Omron Sysmac Studio project AGV_Mohn (Sysmac Studio 1.54.0.19, StandardProject)
(* New standard program for Dahl vehicles, equal bufferlane FB as Alpma *)

# Controller AGV_Mohn: NX1P2-9024DT1 version 1.46
Units and slaves: Node1 : NX-ECC203 (E001); Unit 2 : NX-SID800 (N3_N2); Unit 3 : NX-SID800 (N3_N3); Unit 4 : NX-SOD400 (N3_N4); Unit 5 : NX-SOD400 (N3_N5); Unit 6 : NX-SOH200 (N3_N6); Unit 7 : NX-DA3605 (N1); Unit 8 : NX-AD2203 (N3_N8); Unit 9 : NX-EC0122 (N3); Unit 1 : NX-OD3268 (N2_N1)
Task PrimaryTask (priority 4, period or condition 2000): Communication, AGV_Control, Manual_control, Navitrol, IO_List
Library MQTT 0.45_b14 0.0.45 (contents left out)
Library WewoNavitrol 1.0.2 (contents left out)

TYPE MQTTval : STRUCT
    topic : string[128];
    currentValue : STRING[512];
    sentValue : STRING[512];
END_STRUCT END_TYPE
TYPE Node_State : (STATE_Offline := 0, STATE_Online := 1, STATE_Stop := 2); END_TYPE
TYPE Navitrol_ProductionData_struct : STRUCT
    ProtocolVersion : UINT;  (* Navitrol protocol version; offset 0.0 *)
    Message_ID : UINT;  (* Message ID (3202); offset 2.0 *)
    Message_length : UDINT;  (* Message length in bytes (48 bytes); offset 4.0 *)
    OID_external : UDINT;  (* offset 8.0 *)
    OID_sent : UDINT;  (* offset 12.0 *)
    OID_active : UDINT;  (* offset 16.0 *)
    Item_type : UDINT;  (* offset 20.0 *)
    Pickup_ID : UDINT;  (* offset 24.0 *)
    Target_ID : UDINT;  (* offset 28.0 *)
    Order_status : UINT;  (* offset 32.0 *)
    In_Production : UINT;  (* offset 34.0 *)
END_STRUCT END_TYPE
TYPE Navitrol_TargetDetectionStatus_struct : STRUCT
    ProtocolVersion : UINT;  (* offset 0.0 *)
    Message_ID : UINT;  (* offset 2.0 *)
    Message_length : UDINT;  (* offset 4.0 *)
    DetectionMode : BYTE;  (* offset 8.0 *)
    TargetFount : BYTE;  (* offset 9.0 *)
    TargetReached : BYTE;  (* offset 10.0 *)
    TargetWithinSafetyDistance : BYTE;  (* offset 11.0 *)
    TargetX : REAL;  (* offset 12.0 *)
    TargetY : REAL;  (* offset 16.0 *)
    TargetAngle : REAL;  (* offset 20.0 *)
    PalletIDBeingDetected : DWORD;  (* offset 24.0 *)
    NumberOfReflectorsBeingDetected : UINT;  (* offset 28.0 *)
    FoundPallet’sID : UINT;  (* offset 30.0 *)
    ReservedField1 : UDINT;  (* offset 32.0 *)
    ReservedField2 : UDINT;  (* offset 36.0 *)
    ReservedField3 : UDINT;  (* offset 40.0 *)
    ReservedField4 : UDINT;  (* offset 44.0 *)
    ReservedField5 : UDINT;  (* offset 48.0 *)
END_STRUCT END_TYPE
TYPE Navitrol_ErrorWithLevel_Struct : STRUCT
    ProtocolVersion : UINT;  (* offset 0.0 *)
    Message_ID : UINT;  (* offset 2.0 *)
    Message_Length : UDINT;  (* offset 4.0 *)
    LevelOfHighestError : UINT;  (* offset 8.0 *)
    Reserved1 : UDINT;  (* offset 10.0 *)
    ErrorCount : UDINT;  (* offset 14.0 *)
    ErrorList : ARRAY[0..15] OF Navitrol_ErrorWithLevel_Error_Struct;  (* offset 18.0 *)
END_STRUCT END_TYPE
TYPE Navitrol_ErrorWithLevel_Error_Struct : STRUCT
    ErrorCode : UDINT;  (* offset 0.0 *)
    ErrorLevel : UDINT;  (* offset 4.0 *)
    Reserved2 : UINT;  (* offset 8.0 *)
END_STRUCT END_TYPE
TYPE Actuator_Selection : (Neither := 0, Front := 1, Rear := 2, Both := 3); END_TYPE
TYPE LED_Colour : (LED_Red := 0, LED_Orange := 1, LED_Yellow := 2, LED_Green := 3, LED_Cyan := 4, LED_Blue := 5, LED_Magenta := 6, LED_White := 7); END_TYPE
TYPE MES_Data_struct : STRUCT  (* MES data word *)
    Heartbeat_out : BOOL;  (* Feedback state of received heartbeat; offset 0.0 *)
    Idle : BOOL;  (* AGV in idle state; offset 0.1 *)
    Emergency : BOOL;  (* AGV in emergency state (stop state); offset 0.2 *)
    Obstacle : BOOL;  (* Obstacle in scanner warning; offset 0.3 *)
    Manual : BOOL;  (* AGV in manual ControlModeLift; offset 0.4 *)
    Loaded : BOOL;  (* AGV loaded or override active; offset 0.5 *)
    Actuator : BOOL;  (* Actuator active; offset 0.6 *)
    Charging : BOOL;  (* AGV being charged; offset 0.7 *)
    ObstacleStop : BOOL;  (* AGV stopped for obstacle; offset 1.0 *)
    ObstacleEstop : BOOL;  (* Object in sfety field; offset 1.1 *)
    Overhang : BOOL;  (* Overhang object sees object; offset 1.2 *)
    DoorState : BOOL;  (* Doorstatus, 1=ok; offset 1.3 *)
    ForkCollision : BOOL;  (* Fork collision status; offset 1.4 *)
    LiftWarning : BOOL;  (* Lift in warning state (unoperational); offset 1.5 *)
    LiftAuto : BOOL;  (* Lift busy with MES command; offset 1.6 *)
    DockingActive : BOOL;  (* AGV in docking state; offset 1.7 *)
END_STRUCT END_TYPE
TYPE Lift_Req_State : (Lift_Off := 0, Lift_Up := 1, Lift_Down := 2); END_TYPE
TYPE MQTT_Actuator_Request_struct : STRUCT  (* x coordinante of target *)
    Target_X : REAL;  (* y coordinante of target *)
    Target_Y : REAL;  (* Target position ID *)
    Distance : REAL;  (* Distance from target from inner and outer commands *)
    Height_Inner : INT;  (* Near target actuator height *)
    Height_Outer : INT;  (* Far from target actuator height *)
    Cargo_Required : BOOL;  (* Height_Inner needs cargo if true *)
END_STRUCT END_TYPE
TYPE Webinterface_Reply_struct : STRUCT
    State : BYTE;  (* offset 0.0 *)
    Timing : UINT;  (* offset 1.0 *)
    Version : STRING[5];  (* offset 3.0 *)
    Teaching : BYTE;  (* offset 8.0 *)
    V : REAL;  (* offset 9.0 *)
    X : REAL;  (* offset 13.0 *)
    Y : REAL;  (* offset 17.0 *)
    H : REAL;  (* offset 21.0 *)
    Level : BYTE;  (* offset 25.0 *)
    Pos_Conf : REAL;  (* offset 26.0 *)
    Error : BYTE;  (* offset 30.0 *)
    Nav_State : BYTE;  (* offset 31.0 *)
    SoC : REAL;  (* offset 32.0 *)
    Rem_Address : STRING[15];  (* offset 36.0 *)
    Mach_Type : BYTE;  (* offset 51.0 *)
    Omni_Steer : BYTE;  (* offset 52.0 *)
    Sector_Max : REAL;  (* offset 53.0 *)
    Sector_Min : REAL;  (* offset 57.0 *)
    Deadband : REAL;  (* offset 61.0 *)
    On_Route : BYTE;  (* offset 65.0 *)
    Fatal_Active : BYTE;  (* offset 66.0 *)
    Mach_ID : BYTE;  (* offset 67.0 *)
    Token : UINT;  (* offset 68.0 *)
    AgvLoaded : BYTE;  (* offset 73.0 *)
    Act_Active : BYTE;  (* offset 74.0 *)
    Act_Exist : BYTE;  (* offset 75.0 *)
END_STRUCT END_TYPE
TYPE Navitrol_SetTargetDetectionControlModeLift_struct : STRUCT
    ProtocolVersion : UINT;  (* Navitrol protocol version; offset 0.0 *)
    Message_ID : UINT;  (* Message ID (3202); offset 2.0 *)
    Message_length : UDINT;  (* Message length in bytes (48 bytes); offset 4.0 *)
    TargetDetectionControlModeLift : UINT;  (* Detection ControlModeLift, 0=off, 2=pallet detection; offset 8.0 *)
    PalletsToDetect : UDINT;  (* Bitfield (bit 0=ControlModeLiftl0, bit 1=ControlModeLiftl1, etc.); offset 10.0 *)
    NrOfReflectors : UINT;  (* Number of reflectors used in reflector docking; offset 14.0 *)
    ReflectorWidth : UINT;  (* Width of the used reflectors in mm; offset 16.0 *)
    PatternDetdist0 : UINT;  (* Distances (millimeter) between center of reflectors; offset 18.0 *)
    PatternDetdist1 : UINT;  (* Distances (millimeter) between center of reflectors; offset 20.0 *)
    PatternDetdist2 : UINT;  (* Distances (millimeter) between center of reflectors; offset 22.0 *)
    PatternDetdist3 : UINT;  (* Distances (millimeter) between center of reflectors; offset 24.0 *)
    PatternDetdist4 : UINT;  (* Distances (millimeter) between center of reflectors; offset 26.0 *)
    PatternDetdist5 : UINT;  (* Distances (millimeter) between center of reflectors; offset 28.0 *)
    PatternDetdist6 : UINT;  (* Distances (millimeter) between center of reflectors; offset 30.0 *)
    Reserved1 : UDINT;  (* Reserved bytes; offset 32.0 *)
    Reserved2 : UDINT;  (* Reserved bytes; offset 36.0 *)
    Reserved3 : UDINT;  (* Reserved bytes; offset 40.0 *)
    Reserved4 : UDINT;  (* Reserved bytes; offset 44.0 *)
END_STRUCT END_TYPE
TYPE Navitrol_SaveLogs_struct : STRUCT
    ProtocolVersion : UINT;  (* Navitrol protocol version; offset 0.0 *)
    Message_ID : UINT;  (* Message ID (1007); offset 2.0 *)
    Message_length : UDINT;  (* Message length in bytes (8 bytes); offset 4.0 *)
END_STRUCT END_TYPE
TYPE Navitrol_PauseDrive_struct : STRUCT
    ProtocolVersion : UINT;  (* Navitrol protocol version; offset 0.0 *)
    Message_ID : UINT;  (* Message ID (3006); offset 2.0 *)
    Message_length : UDINT;  (* Message length in bytes (8 bytes); offset 4.0 *)
END_STRUCT END_TYPE
TYPE Navitrol_ResumeDrive_struct : STRUCT
    ProtocolVersion : UINT;  (* Navitrol protocol version; offset 0.0 *)
    Message_ID : UINT;  (* Message ID (3007); offset 2.0 *)
    Message_length : UDINT;  (* Message length in bytes (8 bytes); offset 4.0 *)
END_STRUCT END_TYPE
TYPE Navitrol_AbortDrive_struct : STRUCT
    ProtocolVersion : UINT;  (* Navitrol protocol version; offset 0.0 *)
    Message_ID : UINT;  (* Message ID (3008); offset 2.0 *)
    Message_length : UDINT;  (* Message length in bytes (8 bytes); offset 4.0 *)
END_STRUCT END_TYPE
TYPE Navitrol_SetSpeedLimit_struct : STRUCT
    ProtocolVersion : UINT;  (* Navitrol protocol version; offset 0.0 *)
    Message_ID : UINT;  (* Message ID (3023); offset 2.0 *)
    Message_length : UDINT;  (* Message length in bytes (14 bytes); offset 4.0 *)
    SetRelease : UINT;  (* 1=set limit, 0=release limits; offset 8.0 *)
    Speed : REAL;  (* Speed in m/s; offset 10.0 *)
END_STRUCT END_TYPE
TYPE Navitrol_AbortWithData_struct : STRUCT
    ProtocolVersion : UINT;  (* Navitrol protocol version; offset 0.0 *)
    Message_ID : UINT;  (* Message ID (3033); offset 2.0 *)
    Message_length : UDINT;  (* Message length in bytes (14 bytes); offset 4.0 *)
    StatusControl : Navitrol_AbortControl_struct;  (* Bit field; offset 8.0 *)
    Reserved1 : UINT;  (* offset 10.0 *)
    Reserved2 : UINT;  (* offset 12.0 *)
END_STRUCT END_TYPE
TYPE Navitrol_AbortControl_struct : STRUCT
    EndDriveCompleted : BOOL;  (* 1=drive completed, 0=drive needs to be resend; offset 0.0 *)
    Reserved1 : BOOL;  (* offset 0.1 *)
    Reserved2 : BOOL;  (* offset 0.2 *)
    Reserved3 : BOOL;  (* offset 0.3 *)
    Reserved4 : BOOL;  (* offset 0.4 *)
    Reserved5 : BOOL;  (* offset 0.5 *)
    Reserved6 : BOOL;  (* offset 0.6 *)
    Reserved7 : BOOL;  (* offset 0.7 *)
    Reserved8 : BOOL;  (* offset 1.0 *)
    Reserved9 : BOOL;  (* offset 1.1 *)
    Reserved10 : BOOL;  (* offset 1.2 *)
    Reserved11 : BOOL;  (* offset 1.3 *)
    Reserved12 : BOOL;  (* offset 1.4 *)
    Reserved13 : BOOL;  (* offset 1.5 *)
    Reserved14 : BOOL;  (* offset 1.6 *)
    Reserved15 : BOOL;  (* offset 1.7 *)
END_STRUCT END_TYPE
TYPE Navitrol_RequestDriveCompleted_struct : STRUCT
    ProtocolVersion : UINT;  (* Navitrol protocol version; offset 0.0 *)
    Message_ID : UINT;  (* Message ID (3038); offset 2.0 *)
    Message_length : UDINT;  (* Message length in bytes (10 bytes); offset 4.0 *)
    Request : UINT;  (* 0=none, 1=docking, 2=buffer lane, 3=generic; offset 8.0 *)
END_STRUCT END_TYPE
TYPE Navitrol_SetSpeedArray_struct : STRUCT
    ProtocolVersion : UINT;  (* Navitrol protocol version; offset 0.0 *)
    Message_ID : UINT;  (* Message ID (3028); offset 2.0 *)
    Message_length : UDINT;  (* Message length in bytes (12 bytes); offset 4.0 *)
    SetRelease : UINT;  (* 1=set limit, 0=release limits; offset 8.0 *)
    Speed : UINT;  (* Array index to select; offset 10.0 *)
END_STRUCT END_TYPE
TYPE Navitrol_Errorlist_struct : STRUCT
    ProtocolVersion : UINT;  (* Navitrol protocol version; offset 0.0 *)
    Message_ID : UINT;  (* Message ID (201); offset 2.0 *)
    Message_length : UDINT;  (* Message length in bytes (variable); offset 4.0 *)
    Errcount : UDINT;  (* Amount of errors send (each is an UDINT); offset 8.0 *)
END_STRUCT END_TYPE
TYPE State_Scanner : (SCAN_Clear := 0, SCAN_Warn := 1, SCAN_Stop := 2, SCAN_eStop := 3); END_TYPE
TYPE Error_level_Enum : (Ok := 0 (* No Controller error *), Partial := 2 (* Partial fault level *), Minor := 3 (* Minor fault level *)); END_TYPE
TYPE Navitrol_RequestProductionData_struct : STRUCT
    ProtocolVersion : UINT;  (* offset 0.0 *)
    Message_ID : UINT;  (* offset 2.0 *)
    Message_length : UDINT;  (* offset 4.0 *)
    Activate_sending : UINT;  (* offset 8.0 *)
END_STRUCT END_TYPE
TYPE Pallet_Det_State : (init := 0, assent_PLC := 1, lift_Goes_To_Target := 2, counted_Pallets := 3); END_TYPE
TYPE Palletdetection_Action : (Mes_NotActive := 0, Mes_Active := 1); END_TYPE
TYPE ControlLift : (AGVusesNoLift := 0, Manual := 1, Automatic := 2 (* Controlled by MES *), SemiAutomatic := 3); END_TYPE
TYPE Lane_drop_state : (Idle_drop := 0, Active_drop := 10, Ready_to_drop := 20, Finished_drop := 30); END_TYPE
TYPE Navitrol_TargetDetectionStatusToMes_struct : STRUCT
    TargetFount : STRING[3];
    TargetReached : STRING[3];
    TargetWithinSafetyDistance : STRING[3];
    TargetX : STRING[100];
    TargetY : STRING[100];
    Angle : STRING[100];
END_STRUCT END_TYPE
TYPE MQTT_Errors_struct : STRUCT  (* x coordinante of target *)
    Error1 : STRING[256];
END_STRUCT END_TYPE
TYPE MQTT_Popup_struct : STRUCT  (* x coordinante of target *)
    ScreenLayer : INT;
    Message : STRING[256];
END_STRUCT END_TYPE
TYPE MQTT_Warnings_struct : STRUCT  (* x coordinante of target *)
    Warning1 : STRING[256];
END_STRUCT END_TYPE
TYPE stAnalogSensor : STRUCT
    RAW_VAL : INT;  (* Raw value *)
    OVR_VAL : INT;  (* Max error value *)
    UNDR_VAL : INT;  (* Min error value *)
    SP_MAX : INT;  (* Max setpoint value *)
    SP_MIN : INT;  (* Min setpoint value *)
    BWIRE_VAL : INT;  (* Broken wire value *)
    ALM_BWIRE : BOOL;  (* Broken wire detected *)
    ALM_OVR : BOOL;  (* Sensor over range *)
    ALM_OOR : BOOL;  (* Sensor out of range *)
    ALM_UNDR : BOOL;  (* Sensor under range *)
END_STRUCT END_TYPE
TYPE stBufferError : STRUCT
    CargoSensorBWIRE : BOOL;  (* Ultrasoon cargo distance sensor has broken wire *)
    BufferlaneSensorOOR : BOOL;  (* Laser distance sensor out of range *)
    LiftHeight : BOOL;  (* Lift height check when entering bufferlane *)
    StateErrorMES : BOOL;  (* Load not in range, can't be picked in lane *)
END_STRUCT END_TYPE
TYPE stBufferlane : STRUCT
    State : stBufferlaneStatus;  (* Status of bufferlane action *)
    Error : stBufferError;  (* Errors occured in bufferlane *)
END_STRUCT END_TYPE
TYPE stBufferlaneStatus : STRUCT
    ePickSTAT : Lane_pick_state;  (* Pick status *)
    eDropSTAT : Lane_drop_state;  (* Drop status *)
END_STRUCT END_TYPE
TYPE stControl : STRUCT
    NavInProduction : UINT;  (* Navitec in production *)
    NavInManual : BOOL;  (* Navitec in manual state *)
    NavTargetReached : UINT;  (* Navitrol reached target status *)
    NavCust1 : REAL;  (* Special route property in Navithor Tools *)
    NavCust2 : REAL;  (* Special route property in Navithor Tools *)
    NavCust3 : REAL;  (* Special route property in Navithor Tools *)
    NavCust4 : REAL;  (* Special route property in Navithor Tools *)
    NavCust5 : REAL;  (* Special route property in Navithor Tools *)
    BufferAction : INT;  (* Pick or drop action determined by MES *)
    BufferReleaseHold : BOOL;  (* Release AGV determined by MES *)
    AGVloaded : BOOL;  (* AGV is loaded *)
    AGVdir : BOOL;  (* 0 = fwdDirection of AGV *)
    AGVstandstill : BOOL;  (* AGV standstill *)
    CargoRequired : BOOL;  (* Cargo required *)
    ClientConnected : BOOL;  (* MQTT client connected *)
    ResetButton : BOOL;  (* Reset errors by operator *)
END_STRUCT END_TYPE
TYPE Lane_pick_state : (Idle_pick := 0, Active_pick := 10, Ready_to_lower_lift_pick := 20, Ready_to_pick := 30, Finished_pick := 40); END_TYPE
TYPE Lane_state_MES : (Idle := 0, Picking_Active := 10, Picking_Drive_In := 20, Picking := 30, Picking_Finished := 40, Dropping_Active := 50, Dropping := 60, Dropping_Finished := 70); END_TYPE
TYPE stClampError : STRUCT  (* Error handling for customer Alpma *)
    ClampSensorBWIRE : BOOL;  (* One of clamp sensor broken wire *)
END_STRUCT END_TYPE
TYPE stOverhang : STRUCT
    UsesPF : BOOL;  (* Pepperl and Fuchs sensor *)
    UsesSICK : BOOL;  (* SICK sensor *)
    DetectedPF : BOOL;  (* PFuchs sensor detect signal *)
    DetectedSICK : BOOL;  (* SICK sensor detect signal *)
END_STRUCT END_TYPE
TYPE stClamp : STRUCT
    IO : stClampIO;
    CargoClamped : BOOL;  (* Cargo is clamped *)
END_STRUCT END_TYPE
TYPE stClampIO : STRUCT
    Load1 : BOOL;  (* Switch NC sensor 1 in clamp *)
    Load2 : BOOL;  (* Switch NC sensor 2 in clamp *)
    Attached : BOOL;  (* Feedback clamp is attached *)
END_STRUCT END_TYPE

VAR_GLOBAL
    ClientConnected : BOOL;  (* MQTT client connected *)
    Mqtt_values : ARRAY[0..32] OF MQTTval;  (* Address:; [0] will; [1] liftHeight; [2] load; [3] safety; [4] eStopButton; [5] scanner1; [6] scanner2; [7] scanner3; [8] docking; [9] manualDrive; [10] manualLift; [11] brakeRelease; [12] charging; [13] cancelRequest; [14] cancelConfirm; [15] forkCollision *)
    Stations_State : Node_State;
    MES_State : Node_State;
    MES_Target : MQTT_Actuator_Request_struct;  (* MES actuator request by MQTT *)
    MES_PalletDetection : Palletdetection_Action;
    AGVusesRS232 : BOOL;
    AGV_Init : UINT := 0;  (* A runonce function to load values into registers *)
    Dir_Encoder1 : BOOL;  (* 0=Forward *)
    Brake_Override_Switch : BOOL;  (* Manual override switch *)
    Manual_ControlModeLift : BOOL;
    AGV_Docking : BOOL;  (* Safety reports AGV in docking ControlModeLift; at ECAT://node#[1,1]/Docking_Active *)
    Reset_Flag : BOOL;  (* Reset function called *)
    Navitrol_Tag : Navitrol_Status_TagV4_sec_struct;  (* Navitrol tag status message *)
    ToChargerTag : UDINT;  (* Virtual tag id *)
    ChargerTag : UDINT;  (* Tag ID for chargers *)
    Standstill : BOOL;  (* DoubleCheck for 0 speed *)
    Charge_Relay : BOOL;  (* Enable contact power *)
END_VAR
VAR_GLOBAL CONSTANT
    RS232_BoardID : _sOPTBOARD_ID := (SlotNo := 1, IPAdr := [5(16#0)]);  (* Board ID *)
END_VAR
VAR_GLOBAL
    ENC1_Dir_Raw : BOOL;  (* Value from enocder slice; at ECAT://node#[1,9]/Ch1 Encoder Counter Status/Ch1 Count Direction Flag *)
    ENC1_Dir : BOOL;
    Scanner_Stop : BOOL;  (* object in safety field *)
    Pump_Ok : BOOL;  (* Pump system ok *)
    Estop_Out : BOOL;  (* E-Stop has been pressed and not yet reset; at ECAT://node#[1,1]/Estop_Out *)
    Motor_Ok : BOOL;  (* Motor power active *)
    PLC_status : PLC_Status_Struct;  (* PLC status message *)
    Motor_Power_1 : BOOL;  (* Power relay 1 coil; at ECAT://node#[1,6]/Standard Input 1st Byte/So00 Monitor Value *)
    Motor_Power_2 : BOOL;  (* Power relay 2 coil; at ECAT://node#[1,6]/Standard Input 1st Byte/So01 Monitor Value *)
    Pump_Power_1 : BOOL;
    Pump_Power_2 : BOOL;
    Warning_ActuatorTime : BOOL;  (* Lift action took too long *)
    Brake_release : BOOL;  (* Brakes manual release *)
    ENC1_Speed : REAL;  (* Encoder speed in m/s *)
    Navitrol_status : Navitrol_Status_Struct;  (* Navitrol status message *)
    RotPerMin : REAL;  (* Encoder rotation per minute *)
    ENC1_Rate : UDINT;  (* Measured speed in pulses; at ECAT://node#[1,9]/Ch1 Pulse Rate *)
    AGVusesActuator : BOOL;  (* True makes sure status message is updated in the actuator section *)
    AGVusesSteering : BOOL;  (* AGV uses a steering wheel to manouver, set to 0 for differential drive *)
    AGVhasHandheld : BOOL;  (* AGV can be controlled using remote control *)
    AnalogLoad : BOOL;  (* AGV uses an analog sensor for load detection *)
    AGV_MaxSpeed : REAL;  (* Max speed in m/s *)
    NavitrolArrayLimit : BOOL;  (* Use navitrol speed array *)
    NavitrolSpeedLimit : BOOL;  (* use navitrol speed limit *)
END_VAR
VAR_GLOBAL RETAIN
    MachineID : INT;  (* Machine ID from navithor & MES *)
END_VAR
VAR_GLOBAL
    Navitrol_IP : STRING[256] := '';  (* Navigation controller *)
    Navitrol_TX_Port : UINT := 0;  (* TCP server port *)
    Navitrol_RX_Port : UINT := 0;  (* TCP listen port *)
    Navitrol_ManualSection_Enabled : BOOL;  (* Send manual section to Navitrol *)
    Navitrol_ErrorSection_Enabled : BOOL;  (* Send error messages to Navitrol *)
    Navitrol_InputSection_Enabled : BOOL;  (* Send input section to Navitrol *)
    Navitrol_LaserSection_Enabled : BOOL;  (* Send laser scanner section to Navitrol *)
    RequestGeneralSection : BOOL;  (* Ask for the general section (ID=1) from navitrol status *)
    RequestHoldSection : BOOL;  (* Ask for the hold section (ID=2) from navitrol status *)
    RequestVirtualTagSection : BOOL;  (* Ask for the virtual tag section (ID=3) from navitrol status *)
    RequestComingGoingSection : BOOL;  (* Ask for the 'Coming from, going to' section (ID=4) from navitrol status *)
    RequestCustomAtributeSection : BOOL;  (* Ask for the custom atribute section (ID=6) from navitrol status *)
    RequestWarningSection : BOOL;  (* Ask for the warning zone section (ID=7) from navitrol status *)
    RequestOutputsSection : BOOL;  (* Ask for the output section (ID=8) from navitrol status *)
    RequestBatterySection : BOOL;
    RequestDriveInfoSection : BOOL;
    RequestDistanceInfoSection : BOOL;
    NrOfSections : UINT := 0;  (* Amount of requested sections *)
    Sections : ARRAY[1..10] OF UINT;  (* Array for requested sections *)
    Navitrol_ActSection_Enabled : BOOL;  (* Send actuator section to Navitrol *)
    PLC_act : PLC_Act_Sec_Struct;
    Lift_Bot_Pos : BOOL;
    Lift_Top_Pos : BOOL;
    MessageLength : UDINT;  (* Tx message length in bytes *)
    RequestSteeringAngleSection : BOOL;  (* Ask for the steering angle section (ID=9) from navitrol status, sets with AGVusesSteering *)
    ActuatorAction : BOOL;  (* Remove power from drive motor *)
    Reset_Button : BOOL;  (* Reset input button *)
    HMI_Input0 AT %0.00 : BOOL;  (* RESET; published *)
    Safe_Reset_button : BOOL;  (* Reset button status for safety; at ECAT://node#[1,1]/Reset_Button *)
    Rel_Spd_Nav1 : INT;  (* Navitrol relative vehicle speed; at ECAT://node#[1,1]/Speed_Nav *)
    Abs_Spd_Enc1 : INT;  (* Encoder 1 absolute wheel speed *)
    Steering_Cos_Rad : REAL;  (* Cosine from target angle in Rad *)
    Navitrol_Steer : Navitrol_Status_Steering_Sec_Struct;
    Rel_Spd_Enc1 : INT;  (* Encoder relative vehicle speed; at ECAT://node#[1,1]/Speed_Enc_Rel *)
    Comp_Rel_Spd_Enc1 : INT;  (* Compensated relative enocder speed; at ECAT://node#[1,1]/Speed_Enc *)
    Dir_Navitrol1 : BOOL;  (* 0=Forward *)
    OptionalFieldReq : INT;  (* Special field selection; at ECAT://node#[1,1]/OptionalFieldReq *)
    Navitrol_SpeedUpdate : BOOL;  (* Navitrol should use a different speed setting *)
    SetNavitrolSpeedLimit : BOOL;  (* Send true to use speed limiter *)
    SpeedArray : UINT;  (* Array selection (0..4) *)
    SpeedLimit : REAL;  (* Max speed in m/s for limiter message *)
    Board_Detected : BOOL;  (* Sensor detects fork board *)
    Scanner_Slowdown : BOOL;  (* object in slowdown field *)
    Safe_Scanner_Slowdown : BOOL;  (* Slowdown to 0 field status to safety; at ECAT://node#[1,1]/Scanner_slowdown *)
    Error_Fork_Object : BOOL;  (* Fork object detection triggered *)
    Estop_requested : BOOL;  (* Request uncontrolled stop from safety; at ECAT://node#[1,1]/Estop_Request *)
    Scan1_Warn : BOOL;  (* Front right warning field *)
    Scanner_Warning : BOOL;  (* object in outer field *)
    Warning_SlowedByObstacle : BOOL;  (* Object detected in outer field while moving *)
    Scan1_Slow : BOOL;  (* Front right stop field *)
    Warning_StoppedByObstacle : BOOL;  (* Object detected in slowdown field *)
    Warning_Active : BOOL;  (* A warning is active *)
    Error_Active : BOOL;  (* A error is active *)
    HMI_Input7 AT %0.07 : BOOL;  (* Buzzer button *)
    Buzzer : BOOL;  (* Audio output *)
    PLC_Navitrol_laserscanners : PLC_Navitrol_Status_laserscanner_struct;  (* PLC to Navitrol laserscanner section *)
    Warning_StopNavitrol : BOOL;  (* AGV keeps navitrol stopped *)
    Right_door_closed : BOOL;  (* Cover is closed *)
    Left_door_closed : BOOL;  (* Cover is closed *)
    Front_door_closed : BOOL;  (* Cover is closed *)
    Warning_Cover_Open : BOOL;  (* One or more covers are not closed *)
    Lift_pump : BOOL;  (* Enables hydraulic pump *)
    StopRequest : BOOL;  (* Request controlled stop from safety PLC; at ECAT://node#[1,1]/StopRequest *)
    Update_Navitrol : BOOL;  (* Update navitrol asap *)
    LED_Reset : BOOL;  (* Indicator light *)
    LED_Left : BOOL;  (* Disable left LED bar *)
    LED_Mid1 : BOOL;  (* Disable middle-left LED bar *)
    LED_Right : BOOL;  (* Disable right LED bar *)
    LED_Mid2 : BOOL;  (* Disable middle-right LED bar *)
    Navitrol_DriveInfo : Navitrol_Status_DriveorderInfo_sec_struct;  (* Driveinfo section *)
    Blue_spot1 : BOOL;  (* Front facing Bluespot *)
    Blue_spot2 : BOOL;  (* Rear facing Bluespot *)
    Manual_Navitrol : BOOL;  (* Navitrol in manual state *)
    LED_R : INT;
    LED_G : INT;
    LED_B : INT;
    Navitrol_Battery : Navitrol_Status_Battery_struct;  (* Battery status from navitrol *)
    MES_Out_Ack AT %20.0 : BOOL;  (* Heartbeat that should change every second *)
    MES_Battery AT %20.8 : SINT;
    MES_InProd AT %20.1 : BOOL;  (* AGV in production in Navithor *)
    MES_AGVstatus AT %253 : MES_Data_struct;  (* Word for AGV status *)
    Manual_mode_switch : BOOL;  (* Manual ControlModeLift hardware switch *)
    Warning_NoPallet : BOOL;
    Warning_Lift_NOK : BOOL;  (* Lift sensor not in valid range *)
    MES_Height_Act AT %254 : UINT;  (* Actual height feedback for MES *)
    MES_MID0 AT %20.2 : BOOL;
    MES_MID1 AT %20.3 : BOOL;
    HMI_Input4 AT %0.04 : BOOL;  (* Force docking Mode; published *)
    HMI_Output0 AT %2.00 : BOOL;  (* Show RESET; published *)
    HMI_Output7 AT %2.07 : BOOL;  (* Lid; published *)
    HMI_Input3 AT %0.03 : BOOL;  (* Brake release; published *)
    HMI_Input6 AT %0.06 : BOOL;  (* Silent Mode; published *)
    HMI_Output6 AT %2.06 : BOOL;  (* Silent state; published *)
    HMI_Output9 AT %2.09 : BOOL;  (* Docking state; published *)
    HMI_Output5 AT %2.05 : BOOL;  (* HMI red fork sensors *)
    HMI_Output4 AT %2.04 : BOOL;  (* HMI all clear *)
    HMI_Int2 AT %12 : INT;  (* Front scanner; published *)
    HMI_Int3 AT %13 : INT;  (* Rear Scanner; published *)
    HMI_Int4 AT %14 : INT;  (* Estop state; published *)
    HMI_LED AT %3 : INT;  (* LED colour; published *)
    HMI_Int0 AT %10 : INT;  (* Battery level %; published *)
    HMI_Int1 AT %11 : INT;  (* Position confidence %; published *)
    Scan1_Stop : BOOL;  (* Front right safety scanner status; at ECAT://node#[1,2]/Standard Input 1st Word/Si02 Logical Value *)
    Estop_Channel1 : BOOL;  (* Emergency stop status; at ECAT://node#[1,2]/Standard Input 1st Word/Si00 Logical Value *)
    RM_Estop : BOOL;  (* Remote E-stop  state *)
    HMI_Int5 AT %15 : INT;  (* Machine ID; published *)
    HMI_Int6 AT %16 : INT;  (* HMI height feedback; published *)
    HMI_Int9 AT %19 : INT;  (* Lift max value; published *)
    Error_MotorPower : BOOL;  (* Error in motor feedback; at ECAT://node#[1,1]/Error_MotorEDM *)
    Error_PumpPower : BOOL;  (* Error in pump feedback *)
    Error_Navitrol : BOOL;  (* Navitrol reports an error *)
    Fork_bump_det_1 : BOOL;  (* Fork tip sensor *)
    Fork_bump_det_2 : BOOL;  (* fork tip sensor *)
    WarningCount : USINT := 0;  (* Amount of active warnings counter *)
    PLC_Warn_Array : array[0..4] of PLC_Warn_struct;  (* PLC warning list to send to Navitrol *)
    Warning_TableLift_Without_load : BOOL;  (* Table has been ordered to rise without load present *)
    Warning_TableDrop_Without_Load : BOOL;  (* Table has been ordered to lower without load *)
    Warning_TableLoad_Lost : BOOL;  (* Lost tabel load while lift was high *)
    HMI_Warning1 AT %135 : UINT;  (* Error code for 1st warning; published *)
    HMI_WarningText1 AT %140 : INT;
    HMI_Warning2 AT %136 : UINT;  (* Error code for 2nd warning; published *)
    HMI_WarningText2 AT %144 : INT;
    HMI_Warning3 AT %137 : UINT;  (* Error code for 3rd warning; published *)
    HMI_WarningText3 AT %148 : INT;
    HMI_Warning4 AT %138 : UINT;  (* Error code for 4th warning; published *)
    HMI_WarningText4 AT %152 : INT;
    HMI_Warning5 AT %139 : UINT;  (* Error code for 5th warning; published *)
    HMI_WarningText5 AT %156 : INT;
    ErrorCount : USINT := 0;  (* Amount of active errors counter *)
    Docking_error : BOOL;
    PLC_Error_Array : array[0..4] of PLC_Error_struct;  (* PLC error list to send to Navitrol *)
    SpeedError : BOOL;  (* Error in safety speedcheck; at ECAT://node#[1,1]/SpeedErrorStandard *)
    ErrorIndex : USINT;
    HMI_Error1 AT %50 : UINT;  (* Error code for 1st error; published *)
    HMI_ErrorText1 AT %60 : INT;
    HMI_Error2 AT %51 : UINT;  (* Error code for 2nd error; published *)
    HMI_ErrorText2 AT %64 : INT;
    HMI_Error3 AT %52 : UINT;  (* Error code for 3rd error; published *)
    HMI_ErrorText3 AT %68 : INT;
    HMI_Error4 AT %53 : UINT;  (* Error code for 4th error; published *)
    HMI_ErrorText4 AT %72 : INT;
    HMI_Error5 AT %54 : UINT;  (* Error code for 5th error; published *)
    HMI_ErrorText5 AT %76 : INT;
    Lift_valve : BOOL;  (* Opens hydraulic lift valve *)
    Lift_Prop_Speed : INT;  (* Proportional speed to lift controller *)
    HMI_Input5 AT %0.05 : BOOL;  (* Lift override; published *)
    HMI_Input1 AT %0.01 : BOOL;  (* UP; published *)
    HMI_Input2 AT %0.02 : BOOL;  (* DOWN; published *)
    HMI_Int7 AT %17 : INT;  (* Manual set height; published *)
    Rm_ManDown : BOOL;
    Rm_ManUp : BOOL;
    InProd : BOOL;  (* AGV in production *)
    Navitrol_act : Navitrol_Status_Act_Sec_Struct;
    PumpPower : BOOL;  (* Pump has power; at ECAT://node#[1,1]/PumpPower *)
    Load1 : BOOL;  (* Load sensor 1 *)
    Load2 : BOOL;  (* Load sensor 2 *)
    HMI_Int8 AT %18 : INT;  (* Lift min value; published *)
    N3_N3_Si02 : BOOL;  (* End stop switch for lift; at ECAT://node#[1,3]/Standard Input 1st Word/Si02 Logical Value *)
    Warning_Cargo_NOK : BOOL;  (* Lift action with invalid cargo *)
    TCPReady : BOOL;  (* TCP communication available *)
    RequestDriveReady : BOOL;  (* Target reached *)
    DriveType : UINT;  (* Request ready tpe *)
    Lift_Height_Raw : INT;  (* Encoder value; at ECAT://node#[1,8]/Ch1 Analog Input Value *)
    Navitrol_DistanceInfo : Navitrol_Status_DistanceToTarget_sec_struct;  (* Driveorder information *)
    MES_Height_Req AT %21 : UINT;  (* Desired height from MES *)
    Navitrol_FromTo : Navitrol_Status_FromTo_Sec_struct;
    RM_FR1 : INT;  (* Remote Forward/Reverse channel 1 *)
    RM_Center : INT;  (* Remote center tap *)
    RM_LR1 : INT;  (* Remote Left/Right channel 1 *)
    IPC_Driving_active AT %252 : BOOL;  (* Activate HTTP requests; published *)
    IPC_Driving_x AT %250 : INT;  (* x value to IPC; published *)
    IPC_Driving_y AT %251 : INT;  (* y value to IPC; published *)
    RM_Switch : INT;  (* Remote joystick switch (digital) *)
    RemoteButtonPressed : BOOL;  (* Joystick button is pressed *)
    RM_Dwn : INT;  (* Remote lift down button *)
    RM_Up : INT;  (* Remote lift up button *)
    Remote_Present : BOOL;
    HMI_Input10 AT %0.10 : BOOL;  (* Activate Remote control; published *)
    Error_Remote : BOOL := False;  (* Center tap voltage too low, no remote connected *)
    Navitrol_gen : Navitrol_Status_General_Sec_Struct;  (* Navitrol general message *)
    PLC_Navitrol_input : Navitrol_Status_inputs_struct;  (* PLC to navitrol input values *)
    NumBytes : UINT := 0;  (* Number of bytes in virtual IO (max32) *)
    NumInts : UINT := 0;  (* Number of integers in virtual IO (max32) *)
    NumFloats : UINT := 0;  (* Number of floats in virtual IO (max32) *)
    Navitrol_RemoteControlSection_Enabled : BOOL;
    Navitrol_Drivecontrol_Enabled : BOOL;
    Navitrol_PLC_Battery_Enabled : BOOL;
    NavitrolPause : BOOL;  (* Request navitrol to pause drive *)
    NavitrolResume : BOOL;  (* Request navitrol to resume drive order *)
    SendTargetDetectionSettings : BOOL;  (* send message 3202 to navitrol *)
    NavitrolAbort : BOOL;  (* Request navitrol to abort drive *)
    SafetyFieldNumber : INT;  (* Active field ID; at ECAT://node#[1,1]/ActiveFieldID *)
    Scan2_Stop : BOOL;  (* Front left safety scanner status; at ECAT://node#[1,2]/Standard Input 1st Word/Si04 Logical Value *)
    Motor_EDM_1 : BOOL;  (* Power relay 1 feedback; at ECAT://node#[1,3]/Standard Input 2nd Byte/Si00 Status *)
    Motor_EDM_2 : BOOL;  (* Power relay 2 feedback; at ECAT://node#[1,3]/Standard Input 2nd Byte/Si01 Status *)
    Scan3_Stop : BOOL;  (* Fork safety scanner status; at ECAT://node#[1,2]/Standard Input 1st Word/Si06 Logical Value *)
    Zone1 : BOOL;  (* Scanner zone select 1; at ECAT://node#[1,4]/Standard Input 1st Byte/So00 Monitor Value *)
    zone2 : BOOL;  (* Scanner zone select 2; at ECAT://node#[1,4]/Standard Input 1st Byte/So01 Monitor Value *)
    Zone3 : BOOL;  (* Scanner zone select 3; at ECAT://node#[1,4]/Standard Input 1st Byte/So02 Monitor Value *)
    Zone4 : BOOL;  (* Scanner zone select 4; at ECAT://node#[1,4]/Standard Input 1st Byte/So03 Monitor Value *)
    Zone5 : BOOL;  (* Scanner zone select 5; at ECAT://node#[1,5]/Standard Input 1st Byte/So00 Monitor Value *)
    STO_out : BOOL;  (* Safety torque off signal; at ECAT://node#[1,5]/Standard Input 1st Byte/So02 Monitor Value *)
    BufferLaneSensorDistance : INT;
    Load_Distance : INT;  (* Distance to load; at ECAT://node#[1,8]/Ch2 Analog Input Value *)
    Scan3_Warn : BOOL;  (* Fork warning field *)
    Scan3_slow : BOOL;  (* Fork stop field *)
    Lift_Control_Dir : BOOL;  (* Direction input for lift controller *)
    Indicator_Left : BOOL;  (* Route takes a left turn *)
    Indicator_Right : BOOL;  (* Route takes a right turn *)
    K11 : BOOL;  (* Pump flow direction *)
    K12 : BOOL;  (* Pump flow direction *)
    HMI_Manual AT %2.10 : BOOL;  (* Provide HMI if AGV is in manual state *)
    HMI_Int10 AT %24 : INT;  (* Battery state (enum); published *)
    HMI_MessageCount AT %26 : INT;  (* Total number of warning and error messages; published *)
    SafetyStopped : BOOL;  (* Safety is cutting power; at ECAT://node#[1,1]/SafetyStop *)
    AgvLoaded : BOOL;  (* Object loaded *)
    Scanner1_State : State_Scanner;
    Scanner2_State : State_Scanner;
    Scanner3_State : State_Scanner;
    I00 : BOOL;  (* NX1 input 0; at BuiltInIO://cpu/#0/Input_Bit_00 *)
    I01 : BOOL;  (* NX1 input 1; at BuiltInIO://cpu/#0/Input_Bit_01 *)
    I02 : BOOL;  (* NX1 input 2; at BuiltInIO://cpu/#0/Input_Bit_02 *)
    I03 : BOOL;  (* NX1 input 3; at BuiltInIO://cpu/#0/Input_Bit_03 *)
    I04 : BOOL;  (* NX1 input 4; at BuiltInIO://cpu/#0/Input_Bit_04 *)
    I05 : BOOL;  (* NX1 input 5; at BuiltInIO://cpu/#0/Input_Bit_05 *)
    I06 : BOOL;  (* NX1 input 6; at BuiltInIO://cpu/#0/Input_Bit_06 *)
    I07 : BOOL;  (* NX1 input 7; at BuiltInIO://cpu/#0/Input_Bit_07 *)
    I08 : BOOL;  (* NX1 input 8; at BuiltInIO://cpu/#0/Input_Bit_08 *)
    I09 : BOOL;  (* NX1 input 9; at BuiltInIO://cpu/#0/Input_Bit_09 *)
    I10 : BOOL;  (* NX1 input 10; at BuiltInIO://cpu/#0/Input_Bit_10 *)
    I11 : BOOL;  (* NX1 input 11; at BuiltInIO://cpu/#0/Input_Bit_11 *)
    I12 : BOOL;  (* NX1 input 12; at BuiltInIO://cpu/#0/Input_Bit_12 *)
    I13 : BOOL;  (* NX1 input 13; at BuiltInIO://cpu/#0/Input_Bit_13 *)
    O00 : BOOL;  (* NX1 output 0; at BuiltInIO://cpu/#0/Output_Bit_00 *)
    O01 : BOOL;  (* NX1 output 1; at BuiltInIO://cpu/#0/Output_Bit_01 *)
    O02 : BOOL;  (* NX1 output 2; at BuiltInIO://cpu/#0/Output_Bit_02 *)
    O03 : BOOL;  (* NX1 output 3; at BuiltInIO://cpu/#0/Output_Bit_03 *)
    O04 : BOOL;  (* NX1 output 4; at BuiltInIO://cpu/#0/Output_Bit_04 *)
    O05 : BOOL;  (* NX1 output 5; at BuiltInIO://cpu/#0/Output_Bit_05 *)
    O06 : BOOL;  (* NX1 output 6; at BuiltInIO://cpu/#0/Output_Bit_06 *)
    O07 : BOOL;  (* NX1 output 7; at BuiltInIO://cpu/#0/Output_Bit_07 *)
    O08 : BOOL;  (* NX1 output 8; at BuiltInIO://cpu/#0/Output_Bit_08 *)
    O09 : BOOL;  (* NX1 output 9; at BuiltInIO://cpu/#0/Output_Bit_09 *)
    N10_O00 : BOOL;  (* 2A PNP output 0; at IOBus://unit#1/Output Bit 00 *)
    N10_O01 : BOOL;  (* 2A PNP output 1; at IOBus://unit#1/Output Bit 01 *)
    N10_O02 : BOOL;  (* 2A PNP output 2; at IOBus://unit#1/Output Bit 02 *)
    N10_O03 : BOOL;  (* 2A PNP output 3; at IOBus://unit#1/Output Bit 03 *)
    N11_O00 : BOOL;  (* 2A PNP output 0 *)
    N11_O01 : BOOL;  (* 2A PNP output 1 *)
    N11_O02 : BOOL;  (* 2A PNP output 2 *)
    N11_O03 : BOOL;  (* 2A PNP output 3 *)
    HMI_Input9 AT %0.09 : BOOL;  (* Reset lift *)
    ENC1_Position : DINT;  (* Encoder pulses; at ECAT://node#[1,9]/Ch1 Encoder Present Position *)
    HMI_Unload AT %2.11 : BOOL;
    RequestProductionStatus : BOOL;  (* Request the production status data from Navithor *)
    Navitrol_ProductionStatus : Navitrol_ProductionData_struct;
    Navitrol_TargetDetectionStatus : Navitrol_TargetDetectionStatus_struct;
    Navitrol_ProdDataStatusResult : UINT;  (* 0=not activated, 1=activated *)
    MES_Request_Cancel : BOOL;  (* Operator requests cancel for action *)
    Warning_Mqtt_Client_Error : BOOL;  (* Mqtt client not connected *)
    MES_Cancel_Confirm : BOOL;
    MQTT_enabled : BOOL;  (* MES communication type enabled *)
    Pressure_Sensor_Load : BOOL;
    PalletDetection_state : Pallet_Det_State;
    CountedPallets : INT;
    lift_heavyLoad : BOOL;
    blue : INT;
    RS232_OverhangDetected : BOOL;
    Lift_Controller_Error : BOOL;  (* Lift controller error *)
    Scan2_Warn : BOOL;  (* Front left waring field *)
    Scan2_Slow : BOOL;  (* Front left stop field *)
    Lift_Sensor_Max : BOOL;
    Navitrol_Cust : Navitrol_Status_Custom_sec_struct;  (* Navitrol status, custom attribute *)
    todo : BOOL;
    Zone6 : BOOL;  (* Scanner zone select 6; at ECAT://node#[1,5]/Standard Input 1st Byte/So01 Monitor Value *)
    N3_N3 : BOOL;
    Dir_AGV : BOOL;
    AGV_LaneField : BOOL;  (* at ECAT://node#[1,1]/LaneField_Active *)
    RequestTargetDetectionStatusV2 : BOOL;
    Navitrol_TargetDetectionStatusToMES : Navitrol_TargetDetectionStatusToMes_struct;
    Navitrol_ErrorWithLevel : Navitrol_ErrorWithLevel_Struct;
    MaxSteeringAngleLaneDropping : REAL := 0.17;
    AGVusesLowObstDetect : BOOL;
    HMI_Int11 AT %25 : INT;  (* Start or close popup screen; published *)
    HMI_Int12 AT %27 : INT := 192;  (* IP address Block1 *)
    HMI_Int13 AT %29 : INT := 168;  (* IP address Block2 *)
    HMI_Int14 AT %31 : INT := 8;  (* IP address Block3 *)
    HMI_Int15 AT %33 : INT := 100;  (* IP address Block4 *)
    HMI_String1 AT %80 : STRING[128];  (* Question from MES to answer *)
END_VAR
VAR_GLOBAL RETAIN
    IP_Block1 : INT;
    IP_Block2 : INT;
    IP_Block3 : INT;
    IP_Block4 : INT;
END_VAR
VAR_GLOBAL
    LowObstacleIO : BOOL;  (* Low obstacle sensor detects *)
    MES_Error : MQTT_Errors_struct;  (* MES Error messages by MQTT *)
    MES_Popup : MQTT_Popup_struct;  (* MES Information messages by MQTT *)
    MES_Warning : MQTT_Warnings_struct;  (* MES Warningmessages by MQTT *)
    HMI_Input12 AT %0.12 : BOOL;  (* Confirmation Cancel *)
    HMI_Input11 AT %0.11 : BOOL;
    HMI_Input13 AT %0.13 : BOOL;
    HMI_Int16 AT %34 : INT;  (* MES language update *)
END_VAR
VAR_GLOBAL RETAIN
    MES_Language : INT;
END_VAR
VAR_GLOBAL
    O_LED_B : BOOL;
    O_LED_G : BOOL;
    O_LED_R : BOOL;
    Manual_Mode : BOOL;
    Aout_1 : INT;  (* at ECAT://node#[1,7]/Ch1 Analog Output Value *)
    Aout_2 : INT;  (* at ECAT://node#[1,7]/Ch2 Analog Output Value *)
    Aout_3 : INT;  (* at ECAT://node#[1,7]/Ch3 Analog Output Value *)
    Aout_4 : INT;  (* at ECAT://node#[1,7]/Ch4 Analog Output Value *)
    AGV_Docking_Lane : BOOL;
    AGV_Lane : BOOL;
    AGV_LaneDocking : BOOL;  (* at ECAT://node#[1,1]/Docking_Lane_Active *)
    BufferLaneNavitrol_speed_limiter : BOOL;
    eLaneStateMES : Lane_state_MES;
    HMI_Input14 AT %0.14 : BOOL;  (* Low obstacle HMI *)
    HMI_Output8 AT %2.08 : BOOL;  (* Overhang visualisation *)
    HMI_Output12 AT %2.12 : BOOL;  (* Low obstacle sensor; published *)
    Clamp : stClamp;
    ClampAttached : BOOL;
    NearTarget_No_Load : bool;
END_VAR

(* Program EstopEDM: safety or other program stored in binary form, left out *)

(* Program LaserScanners: safety or other program stored in binary form, left out *)

(* Program SpeedCheck: safety or other program stored in binary form, left out *)

(* FunctionBlock LaserScanners_FB0: safety or other program stored in binary form, left out *)

(* FunctionBlock SpeedCheck_FB: safety or other program stored in binary form, left out *)

(* FunctionBlock SelectorOutputs_FB: safety or other program stored in binary form, left out *)

(* FunctionBlock INT_Conversion: safety or other program stored in binary form, left out *)

(* FunctionBlock ABS_FB: safety or other program stored in binary form, left out *)

(* FunctionBlock SF_InputSelector: safety or other program stored in binary form, left out *)

(* FunctionBlock ScannerZoneSet_Omron_FB: safety or other program stored in binary form, left out *)

(* FunctionBlock ContinuousStop_FB: safety or other program stored in binary form, left out *)

PROGRAM AGV_Control
VAR
    ENC1_Dir_Inv : BOOL;  (* direction correction *)
    Stop_Status : BOOL;
END_VAR
VAR CONSTANT
    NAVITROL_BUFFERLANE : Real := 4;  (* Custom attribute is 4 *)
END_VAR
VAR
    AGV_Accelerating : BOOL;
    ENC1_Acc : REAL;
    debug_chargerelay : BOOL;
END_VAR
VAR CONSTANT
    ChargerDelay_PT : TIME := 2s;  (* Time vehicle must be stationary before charge contacts open *)
    Tag_Charger : UDINT := 55;  (* Tag ID for chargers *)
END_VAR
VAR
    ChargerDelay : TON;
    debug_stoptag : BOOL;
    debug_stop_navitrol : BOOL;  (* stop flag for debug_stoptag *)
    debug_endurance_test : BOOL;  (* Manual endurance test activation *)
    Endurance_timer_reset : BOOL;
    Endurance_ACCTIMER : AccumulationTimer;
END_VAR
VAR RETAIN
    Endurance_Uptime : TIME;  (* Total time in endurance test *)
END_VAR
VAR
    NavitrolCommunication : BOOL;  (* Enable the use of Navitrol communication program *)
    WheelEncPpr : REAL := 15940;  (* Encoder pulses per wheel roatation (PPR * gear ratio) *)
    mPerRot : REAL := 0.722;  (* Distance traveled in m per wheel rotation *)
    ENC1_Speed_ABS : REAL;
    ENC1_Speed_diff : REAL;
    ENC1_Speed_prev : REAL;
    ENC1_Acc_raw : REAL;
    ENC1_Acc_prev : REAL;
    UnloadDistance : DINT;  (* Distance in mm that the AGV shoud moe before raising the lift above scanner level *)
    Max_docking_length : DINT;  (* Max length AGV may drive in docking *)
    SilentMode : BOOL := True;  (* Maintenace mode *)
    AGV_HasDoors : BOOL;  (* AGV has covers that need to be closed *)
    AGV_DockingSpeed : REAL;  (* Max speed for docking ControlModeLift in m/s *)
    NavithorCommunication : BOOL;  (* Enable the use of Navithor communication program *)
    LiftHeightEmpty : INT;  (* Lift height for driving without cargo *)
    LiftHeightLoaded : INT := 400;  (* Lift height for driving with cargo *)
    Lift_Height_Drop : INT;  (* Lift height for drop/pick on the floor *)
    LiftHeightMin : INT;  (* Lift minimal action height *)
    LiftHeightMax : INT;  (* Lift maximal action height *)
    Lift_Height_Docking : INT;  (* Height below which the AGV should be in docking ControlModeLift *)
    Lift_Height_Scale : REAL;
    Lift_Height_Offset : INT;
    DockingTag : UDINT;  (* Tag ID for docking request *)
    NoDockingTag : UDINT;  (* Tag ID for disabling docking ControlModeLift *)
    index : INT;  (* array index *)
END_VAR
VAR RETAIN
    Endurance_Total_meters : ULINT;
    Total_Meters : ULINT;
END_VAR
VAR
    Endurance_Total_meters_start : ULINT;
END_VAR
VAR RETAIN
    Endurance_Total_meters_rel : ULINT;
    Total_Meters_rel : ULINT;
END_VAR
VAR
    Endurance_Total_meters_rel_start : ULINT;
END_VAR
VAR RETAIN
    Endurance_Lift_active_seconds : REAL;
    Lift_active_seconds : REAL;
END_VAR
VAR
    Endurance_Lift_active_seconds_start : REAL;
    Lift_active_time_temp : TIME;
    ActuatorActiveTime : TIME;  (* Time Actuator has been active *)
END_VAR
VAR RETAIN
    Lift_active_hours : REAL;
    Total_Meters_raw : REAL;
    Total_Meters_rel_raw : REAL;
END_VAR
VAR
    Rel_Spd_Enc1_Real : REAL;
    debug_reset : BOOL;
    TP_Reset : TP;
    Navitrol_Speed_REAL : REAL;
    Encoder1_Speed_Real : REAL;
    Encoder1_Speed_Real_ABS : REAL;
    FWD_PT : TIME := 100ms;  (* settle time *)
    FWD_ET : TIME;  (* elapsed time *)
    FWD_TON : TON;
    TON_StandstillSet : TON;
    TON_StandstillReset : TON;
    debug_DockingOn : BOOL;
    HMI_DockingOn : BOOL;  (* HMI requests docking *)
    manual_docking : BOOL;  (* reset button docking request *)
    HMI_DockingOff : BOOL;  (* HMI disables docking *)
    Debug_DockingOff : BOOL;
    Lift_Height : INT;  (* Rounded height in mm *)
END_VAR
VAR CONSTANT
    Tag_Docking : UDINT := 50;  (* Tag ID for docking request *)
END_VAR
VAR
    TON_dockingRequest : TON;
    LiftAtTop : BOOL;  (* Lift close to maximum *)
    LiftHigh : BOOL;  (* Lift above normal height *)
    LiftAtBot : BOOL;  (* Lift in docking range *)
    Navitrol_speed_limiter : BOOL;  (* Reduce Navitrol maximum speed to 0.2m/s *)
    debug_speedset : BOOL;
    debug_speedrelease : BOOL;
    Warning_Signal : BOOL;  (* Sound warning signal *)
    Error_Signal : BOOL;  (* Sound error signal *)
    Audio : BOOL;
    Mute_Audio : BOOL;  (* keep the audio quiet *)
    BuzzerPeriod : TIME;
    BuzzerPulse : TIME;
    PWM_Buzzer : PWM;
    TP_Start_Buzz : TP;
    Navitrol_Warning_Speed : BOOL;  (* Limit speed to 0.3 m/s *)
    TON_WarningAct : TON;
    Hold_By_Actuator : BOOL;  (* AGV has an automated lift action to perform *)
    Reset_Option : BOOL;
    debug_docking_LED : BOOL;
    LED_Scale : INT := 40;  (* LED brightness from 0-150 = 0-100% *)
    PWM_DockingLED : PWM;
    RampDockingLED : Ramp;
    Blink_PT : TIME := 2s;  (* Time blinking should remain active *)
    Blink_Left_TOF : TOF;
    Blink_Right_TOF : TOF;
    IsCharging : BOOL;
    ColourReq : LED_Colour;
    debug_LED : BOOL;
    Colour : LED_Colour;
    debug_Colour : LED_Colour;
    LED_R_Req : INT;
    LED_G_Req : INT;
    LED_B_Req : INT;
    MES_Live : BOOL;  (* MES comm ok *)
    HeartBeat : BOOL;
    TON_MES_Live : TON;
    HMI_Battery : INT;
    MES_MID_temp : USINT;
    MES_MID : USINT;
    TOF_DebugOff : TOF;
    debug_naverror : BOOL;
    debug_forksensor : BOOL;
    Overhang_overruled : BOOL;  (* Overhang detection acknowledged temporary *)
    Pallet_override_active : BOOL;  (* Sensor override by user on HMI *)
    WarningIndex : USINT;
    Lift_Height_Real : REAL;  (* Lift height in mm *)
    Lift_Height_Real_Prev : REAL;  (* Height at last 100ms *)
    Lift_Height_Partial : REAL;  (* Calculation aid *)
    Lift_Rate : REAL;  (* mm per sec *)
    Lift_Allowed : BOOL;
    Lift_Req : Lift_Req_State := Lift_Off;  (* Lift desired direction *)
    Lift_Height_old : INT;
    Lift_NearTarget : BOOL;
    debug_Lift_NearTarget : BOOL;
    debug_ActuatorAction : BOOL;
    LiftPropSpeedUp : INT;
    RampUpLift : Ramp;
    LiftPropSpeedDown : INT;
    Lift_Height_Req : INT := -1;  (* Automatic desired lift height *)
    Lift_dampstart : INT;
    DampenLift : Damp;
    Lift_Prop_Min : INT;
    Lift_Maximal : BOOL;  (* Lift at or above maximal height *)
    Lift_Minimal : BOOL;  (* Lift at or below minimal height *)
    Lift_Set_HMI : BOOL;  (* Auto lift set by HMI *)
    Lift_Action_MES : BOOL;  (* Lift action request from MES *)
    debug_lift : BOOL;
    debug_lift_height : INT;
    debug_lift_allowed : BOOL;
    debug_disableautolift : BOOL;
    Lift_des_speed : INT := 10;  (* Lift desired speed *)
    LiftLimitMax : INT;  (* Final sensor limit *)
    Lift_Req_Min : INT := 85;  (* Lowest value that can be requested *)
    Lift_Req_Max : INT := 2400;  (* Highest value that can be requested *)
    MaxActuatorTime : TIME := 50s;  (* Maximum time the lift may be active *)
    MaxActuatorTime_TON : TON;
    debug_requestdriveready : BOOL;
    Lift_Height_Req_Raw : INT;
    Lift_Minimal_Value : INT := 88;
    Lift_Maximal_Value : INT := 2610;
    Lift_StopRange : REAL;
    debug_TurnLeft : BOOL;
    debug_TurnRight : BOOL;
    Navitrol_Indicator_Right : BOOL;
    Navitrol_Indicator_Left : BOOL;
    LiftPropMax : REAL;  (* max speed *)
    debug_K11 : BOOL;
    debug_valve : BOOL;
    LED_1Hz : BOOL;  (* 1Hz PWM output block *)
    LED_Ramp_Offset : INT := 40;  (* fade offset *)
    LED_Ramp_Period : TIME := 1s;  (* fade time *)
    LED_2Hz : BOOL;  (* 2Hz PWM output block *)
    PWM_BlinkingLED : PWM;
    LED_sync : BOOL;  (* sync flag *)
    temp_speed_up : INT := 7500;
    temp_speed_down : INT := 7500;
    AnalogLoad_Max : REAL;  (* Fork distance for sensor *)
    AnalogLoad_Min : REAL;  (* Minimum value for cargo on fork *)
    AnalogLoad_Cargo_Max : REAL;  (* Valid cargo range *)
    ForkBlocked : BOOL;  (* Analog sensor detects object on fork *)
    Lift_started : BOOL;  (* Lift action in progress *)
    Lift_Near_start : INT;  (* Lift height where damping started *)
    Lift_Rate_Near : REAL;  (* Lift speed during damp action *)
    Lift_Prop_Temp : INT;  (* Calculation aid *)
    LiftNearLimit : INT := 200;  (* Distance from target where damping will start *)
    Lift_Rate_Index : INT;  (* Array index *)
    Lift_Rates : ARRAY[0..9] OF REAL;  (* Average index *)
    Lift_Rate_Partial : REAL;  (* Calculation aid *)
    Lift_AtSpeed : BOOL;  (* Lift reached desired speed *)
    Lift_Rate_Near_Req : REAL;  (* Desired speed during final ramp *)
    Warning_StopNavitrol_TOF : TOF;
    Warning_StopNavitrol_PT : TIME := 250ms;  (* Time to keep navitrol stopped *)
    Warning_StopNavitrol_ET : TIME;  (* elapsed time *)
    debug_MES : BOOL;
    Dropped_Flag : BOOL;  (* AGV has put a cargo down *)
    DroppedPosition : DINT;  (* Encoder puls count at drop point *)
    debug_dropped : BOOL;
    ResetLift : BOOL;
    AGV_AtCargo : BOOL;  (* AGV has reached the cargo *)
    MES_Command_TON : TON;
    MES_Delay : TIME := 500ms;  (* Time for command stabilization *)
    MES_Actuator_Target_UDINT : UDINT;  (* MES target as a UDINT *)
    PLC_Error_Level : Error_level_Enum;  (* Current higest error level *)
    PLC_Error_Level_INT : UINT;  (* 0..3 error level *)
    PLC_Error_Code : DWORD;  (* Code of current active PLC error *)
    FINS_enabled : BOOL;  (* FINS MES communication *)
    InProd_TON : TON;
    InProd_TON_PT : TIME := 5s;  (* Check every time if AGV is in production *)
    Lift_Rate_error : REAL;
    Lift_Prop_Speed_new : INT;
    LiftStopRangeUp : REAL;
    LiftStopRangeDown : REAL;
    Lift_Rate_Partial1 : REAL;
    Lift_Rate_Partial2 : REAL;
    Lift_distance : INT;
    Expected_lift_time_real : REAL;
    Expected_lift_time : TIME;
    ActuatorTime_calculated : BOOL;
    Max_allowed_lift_time : TIME;
    Lift_Rate_diff : REAL;
    ResetPosition : DINT;  (* Encoder position the AGV last moved backwards at *)
    ResetDistance : DINT;  (* Calcuated distance in encoder pulses *)
    LED_Ramp_MinScale : INT := 0;  (* Minimal target *)
    debug_unloadbutton : BOOL;
    Elapsed_lift_time : TIME;
    CurrentTarget : INT;  (* MQTT current action target *)
    Reset_Lift_Busy : BOOL;  (* Prevent MES action until lift has reset *)
    Load_Distance_Real : REAL;
    Load_Distance_Scale : REAL;
    Load_Distance_Offset : INT;
    Start_Position_Drop : DINT;
    Difference_distance_Drop : DINT;
    Difference_Pulses : REAL;
    Distance_Traveled_In_M : REAL;
    Debug_DropCheck : BOOL;
    Distance_Traveled_In_CM : REAL;
    Difference_Between_Load_Drive : REAL;
    Load_Slides_Error : BOOL;
    LiftHeightEmpty_Pallet : INT;
    Lift_Height_Full_Pallet : INT;
    Lift_Height_Max_Empty_Pallet : INT;
    LiftHeightMaxFullPallet : INT;
    Scan : BOOL;
    Palletdetection : PalletDetection_FB;
    Fork_bump_together : BOOL;
    PalletDetection_active : BOOL;
    Lift_At_Target : BOOL;
    PalletDetection_CountedPallets : INT;
    hm : BOOL;
    heavyLoad : SR;
    heavyLoad_reset : BOOL;
    tmp : REAL;
    Overhang_ChargerOverride : BOOL;  (* AGV is aproaching the charger *)
    AGVusesSickOverhang : BOOL;
    Sick_OverhangDetected : BOOL;
    Overhang_PT : TIME;  (* time an object must be within bounds *)
    Overhang_ET : TIME;  (* Elapsed time *)
    Overhang_TON : TON;  (* Overhang stability timer *)
    Reset_Overhang_PT : TIME := 1s;  (* Settle time *)
    Reset_Overhang_ET : TIME;  (* Elapsed time *)
    Reset_Overhang_TON : TON;
    TypeOverhang : INT;
    MES_index : ULINT;
    LiftHeightScale : REAL;  (* Lift height scalar *)
    LiftHeightOffset : INT;  (* Lift height offset *)
    GetLiftHeight : GetCorrectedLiftHeight;
    CorrectedLiftHeight : INT;  (* Current lift height *)
    CorrectedLiftHeight_REAL : REAL;  (* Current lift height real *)
    LiftSpeed : REAL;  (* Current lift speed *)
    LiftSpeedCalculation : CalcLiftSpeed;
    LiftSpeedMax : REAL := 7.0;  (* Maximum lift speed *)
    KpPosUp : REAL := 0.2;  (* P gain for position controller moving up *)
    KpPosDown : REAL := 0.3;  (* P gain for position controller moving down *)
    LiftHeightReq : INT;
    enable : BOOL;
    LiftSpeedSetpoint : REAL;  (* Lift speed setpoint *)
    PositionController : LiftPositionController;
    Speedcontroller : LiftSpeedContoller;
    LiftSpeedMin : REAL := -7.0;  (* Minimuml lift speed *)
    MaxPropAcc : REAL := 50;  (* Maximum proportional acceleration per cycle *)
    KpVel : REAL := 0.4;  (* P gain velocity controller *)
    KiVel : REAL := 0.005;  (* I gain velocity controller *)
    PropStartSpeed : INT := 500;  (* Start proportional speed *)
    ScaledPropSpeed : REAL;  (* Proportional speed scaled to the speed *)
    ControlModeLift : ControlLift;  (* 1=Manual 2=Automatic *)
    LiftHeigtMax : INT;  (* Maximal value empty pallet (in mm from floor) that can be used by fork *)
    ManualControlLift : ManualLift;
    AtTarget : BOOL;  (* Lift at target *)
    LiftReqManual : INT;  (* Lift request manual *)
    LiftRelease : LiftReleaseAtPosition;
    LiftReqAuto : INT;  (* Lift request automatic *)
    LoadingStatus : LiftLoadStatus;
    NearTarget : BOOL;
    LiftPro : REAL;
    MinimalSpeedForError : REAL;  (* minimal speed the lift should reach for not setting an error *)
    LiftReqSemiAuto : INT;
    DroppedFlag : BOOL;
    LiftAutoReset : LiftAutoReset_FB;
    LiftCargoDrag : LiftCargoDrag_FB;
    lif : DINT;
    DistanceTraveledInM : REAL;
    DroppedPositionDrag : DINT;
    CargoDragPT : TIME := 100ms;
    warningCa : BOOL;
    WarningCargoDrag : BOOL;
    CargoDragET : TIME;
    AGVusesHeavyLoadDetection : BOOL;
    TypeWeightDetection : INT;  (* 0= No weight sensor 1= Digital weight sensor 2= Analog weight sensor. *)
    HeavyLoadDetectionMax : BOOL;
    LiftHyeavyLoadDetectionMax : LiftHeavyLoadDetectionMax_FB;
    LiftHeightHeavyLoadMax : INT;  (* Maximum height with heavy load *)
    LiftDetectedHeavyLoad : BOOL;  (* AGV detects heavy load *)
    LiftHyeavyLoadDetection : LiftHeavyLoadDetectionMax_FB;
    LiftLimitMin : INT;
    LaneDropping : Real := 4;
    wa : BOOL;
    MES_LaneDropState : Lane_drop_state;
    slow : BOOL;
    Dir_Enc_TON : TON;
    PWM_TryAgain : PWM;
    Tag_DockingLaneField : UINT := 60;
    ErrorString : STRING[1024];
    SteerTargetAngleABS : REAL;
    Confirmation : BOOL;
    Disable_LowObstacleDetection : BOOL;
    LowObstacle_ChargerOverride : BOOL;
    LowObstacle_PT : TIME;
    SetLowObstacle_TON : TON;
    operatorCancelation : BOOL;
    operatorConfirmation : BOOL;
    Reset_LowObstacle_TON : TON;
    WarningList1 : WarningList;
    DomeLEDs : BOOL;  (* AGV uses Turck dome leds *)
    Scanner_WireReset_Enable : BOOL;
    BufferError : stBufferError;
    Bufferlane : stBufferlane;  (* Bufferlane implementation for customer Alpma *)
    BufferLaneSensorDistance_Max : INT;  (* Max distance of analog sensor, used in bufferlane *)
    BufferLaneSensorDistance_Min : INT;  (* Min distance of analog sensor, used in bufferlane *)
    ErrorList1 : ErrorList_FB;
    fbBufferlane : Bufferlane_FB;
    manual_dockingLane : BOOL;
    MES_LanePickState : Lane_pick_state;
    Warning_BufferlaneCargoClamp : BOOL;
    Warning_BufferlaneHoldAGV : BOOL;  (* Holding AGV while picking or dropping in bufferlane *)
    Warning_BufferlaneLiftHeight : BOOL;
    Warning_BufferlaneSensorOutOfRange : BOOL;
    TON_LanedockingRequest : TON;
    Lift_Height_High : INT;
    AGV_BufferSpeed : REAL;
    Control : stControl;
    ClampError : stClampError;
    stat : BOOL;
    Warning_Overhang : BOOL;
    Overhang : stOverhang;
    fbOverhangDetection : OverhangDET_FB;
    Disable_Overhang : BOOL;
    ove : stOverhang;
    fbLowObstacleDet : LowObstacleDET_FB;
    AGVusesBufferlane : INT;
    CargoSafeLoaded : BOOL;
    NO_OPT_FIELD : INT := 0;
    LANE_FIELD : INT := 4;
    DOCKING_FIELD : INT := 1;
    CHARGER_FIELD : INT := 3;
    MANUAL_FIELD : INT := 2;
    LANE_DOCKING_FIELD : INT := 5;
    Tag_LaneField : UINT;
END_VAR
VAR_EXTERNAL
    AGV_Init : UINT;  (* A runonce function to load values into registers *)
    ENC1_Dir_Raw : BOOL;
    ENC1_Dir : BOOL;
    Scanner_Stop : BOOL;  (* object in safety field *)
    Pump_Ok : BOOL;  (* Pump system ok *)
    Estop_Out : BOOL;
    Motor_Ok : BOOL;  (* Motor power active *)
    PLC_status : PLC_Status_Struct;
    Motor_Power_1 : BOOL;
    Motor_Power_2 : BOOL;
    Pump_Power_1 : BOOL;
    Pump_Power_2 : BOOL;
    Warning_ActuatorTime : BOOL;  (* Lift action took too long *)
    Brake_release : BOOL;
    Manual_ControlModeLift : BOOL;
    Charge_Relay : BOOL;
    ENC1_Speed : REAL;
    Navitrol_status : Navitrol_Status_Struct;
    Navitrol_Tag : Navitrol_Status_TagV4_sec_struct;
    Dir_Encoder1 : BOOL;
    Reset_Flag : BOOL;
    RotPerMin : REAL;  (* Encoder rotation per minute *)
    ENC1_Rate : UDINT;
    AGVusesActuator : BOOL;
    AGVusesSteering : BOOL;
    AGVusesRS232 : BOOL;
    AGVhasHandheld : BOOL;
    AnalogLoad : BOOL;  (* AGV uses an analog sensor for load detection *)
    AGV_MaxSpeed : REAL;  (* Max speed in m/s *)
    NavitrolArrayLimit : BOOL;  (* Use navitrol speed array *)
    NavitrolSpeedLimit : BOOL;  (* use navitrol speed limit *)
    MachineID : INT;
    Navitrol_IP : STRING[256];
    Navitrol_TX_Port : UINT;
    Navitrol_RX_Port : UINT;
    ChargerTag : UDINT;
    ToChargerTag : UDINT;
    Navitrol_ManualSection_Enabled : BOOL;  (* Send manual section to Navitrol *)
    Navitrol_ErrorSection_Enabled : BOOL;  (* Send error messages to Navitrol *)
    Navitrol_InputSection_Enabled : BOOL;  (* Send input section to Navitrol *)
    Navitrol_LaserSection_Enabled : BOOL;  (* Send laser scanner section to Navitrol *)
    RequestGeneralSection : BOOL;
    RequestHoldSection : BOOL;
    RequestVirtualTagSection : BOOL;
    RequestComingGoingSection : BOOL;
    RequestCustomAtributeSection : BOOL;
    RequestWarningSection : BOOL;
    RequestOutputsSection : BOOL;
    RequestBatterySection : BOOL;
    RequestDriveInfoSection : BOOL;
    RequestDistanceInfoSection : BOOL;
    NrOfSections : UINT;
    Sections : ARRAY[1..10] OF UINT;  (* Array for requested sections *)
    Navitrol_ActSection_Enabled : BOOL;
    PLC_act : PLC_Act_Sec_Struct;  (* Navitrol status *)
    Lift_Bot_Pos : BOOL;
    Lift_Top_Pos : BOOL;
    MessageLength : UDINT;  (* Tx message length in bytes *)
    RequestSteeringAngleSection : BOOL;
    ActuatorAction : BOOL;  (* Lift action in progress *)
    Reset_Button : BOOL;
    HMI_Input0 : BOOL;
    Safe_Reset_button : BOOL;
    Rel_Spd_Nav1 : INT;
    Abs_Spd_Enc1 : INT;  (* Encoder 1 absolute wheel speed *)
    Steering_Cos_Rad : REAL;  (* Cosine from target angle in Rad *)
    Navitrol_Steer : Navitrol_Status_Steering_Sec_Struct;
    Rel_Spd_Enc1 : INT;
    Comp_Rel_Spd_Enc1 : INT;
    Dir_Navitrol1 : BOOL;
    Standstill : BOOL;
    OptionalFieldReq : INT;
    Navitrol_SpeedUpdate : BOOL;  (* Navitrol should use a different speed setting *)
    SetNavitrolSpeedLimit : BOOL;
    SpeedArray : UINT;
    SpeedLimit : REAL;
    Board_Detected : BOOL;
    Scanner_Slowdown : BOOL;  (* object in slowdown field *)
    Safe_Scanner_Slowdown : BOOL;  (* Slowdown to 0 field status to safety *)
    Error_Fork_Object : BOOL;  (* Fork object detection triggered *)
    Estop_requested : BOOL;
    Scanner_Warning : BOOL;  (* object in outer field *)
    Warning_SlowedByObstacle : BOOL;  (* Object detected in outer field while moving *)
    Warning_StoppedByObstacle : BOOL;  (* Object detected in slowdown field *)
    Warning_Active : BOOL;  (* A warning is active *)
    Error_Active : BOOL;  (* A error is active *)
    HMI_Input7 : BOOL;
    Buzzer : BOOL;
    PLC_Navitrol_laserscanners : PLC_Navitrol_Status_laserscanner_struct;
    Warning_StopNavitrol : BOOL;  (* AGV keeps navitrol stopped *)
    Right_door_closed : BOOL;
    Left_door_closed : BOOL;
    Front_door_closed : BOOL;
    Brake_Override_Switch : BOOL;
    Warning_Cover_Open : BOOL;  (* One or more covers are not closed *)
    Lift_pump : BOOL;
    StopRequest : BOOL;
    Update_Navitrol : BOOL;
    AGV_Docking : BOOL;
    LED_Reset : BOOL;
    LED_Left : BOOL;
    LED_Mid1 : BOOL;
    LED_Right : BOOL;
    LED_Mid2 : BOOL;
    Navitrol_DriveInfo : Navitrol_Status_DriveorderInfo_sec_struct;
    Blue_spot1 : BOOL;
    Blue_spot2 : BOOL;
    Manual_Navitrol : BOOL;
    LED_R : INT;
    LED_G : INT;
    LED_B : INT;
    Navitrol_Battery : Navitrol_Status_Battery_struct;
    MES_Out_Ack : BOOL;
    MES_Battery : SINT;
    MES_InProd : BOOL;
    MES_AGVstatus : MES_Data_struct;
    Manual_mode_switch : BOOL;
    Warning_NoPallet : BOOL;  (* Cargo sensors did not detect load properly *)
    Warning_Lift_NOK : BOOL;  (* Lift sensor not in valid range *)
    MES_Height_Act : UINT;  (* Actual height feedback for MES *)
    MES_MID0 : BOOL;
    MES_MID1 : BOOL;
    HMI_Input4 : BOOL;
    HMI_Output0 : BOOL;
    HMI_Output7 : BOOL;
    HMI_Input3 : BOOL;
    HMI_Input6 : BOOL;  (* Silent ControlModeLift *)
    HMI_Output6 : BOOL;
    HMI_Output9 : BOOL;
    HMI_Output5 : BOOL;
    HMI_Output4 : BOOL;
    HMI_Int2 : INT;
    HMI_Int3 : INT;
    HMI_Int4 : INT;
    HMI_LED : INT;
    HMI_Int0 : INT;
    HMI_Int1 : INT;
    Estop_Channel1 : BOOL;
    RM_Estop : BOOL;  (* Remote E-stop  state *)
    HMI_Int5 : INT;
    HMI_Int6 : INT;
    HMI_Int9 : INT;
    Error_MotorPower : BOOL;
    Error_PumpPower : BOOL;
    Error_Navitrol : BOOL;  (* Navitrol reports an error *)
    Fork_bump_det_1 : BOOL;
    Fork_bump_det_2 : BOOL;
    WarningCount : USINT;  (* Amount of active warnings counter *)
    PLC_Warn_Array : array[0..4] of PLC_Warn_struct;
    Warning_TableLift_Without_load : BOOL;  (* Table has been ordered to rise without load present *)
    Warning_TableDrop_Without_Load : BOOL;  (* Table has been ordered to lower without load *)
    Warning_TableLoad_Lost : BOOL;  (* Lost tabel load while lift was high *)
    HMI_Warning1 : UINT;
    HMI_WarningText1 : INT;
    HMI_Warning2 : UINT;
    HMI_WarningText2 : INT;
    HMI_Warning3 : UINT;
    HMI_WarningText3 : INT;
    HMI_Warning4 : UINT;
    HMI_WarningText4 : INT;
    HMI_Warning5 : UINT;
    HMI_WarningText5 : INT;
    ErrorCount : USINT;  (* Amount of active errors counter *)
    Docking_error : BOOL;
    PLC_Error_Array : array[0..4] of PLC_Error_struct;  (* PLC error list to send to Navitrol *)
    SpeedError : BOOL;
    ErrorIndex : USINT;
    HMI_Error1 : UINT;
    HMI_ErrorText1 : INT;
    HMI_Error2 : UINT;
    HMI_ErrorText2 : INT;
    HMI_Error3 : UINT;
    HMI_ErrorText3 : INT;
    HMI_Error4 : UINT;
    HMI_ErrorText4 : INT;
    HMI_Error5 : UINT;
    HMI_ErrorText5 : INT;
    Lift_valve : BOOL;
    Lift_Prop_Speed : INT;
    HMI_Input5 : BOOL;
    HMI_Input1 : BOOL;
    HMI_Input2 : BOOL;
    HMI_Int7 : INT;
    Rm_ManDown : BOOL;
    Rm_ManUp : BOOL;
    InProd : BOOL;
    Navitrol_act : Navitrol_Status_Act_Sec_Struct;
    PumpPower : BOOL;
    Load1 : BOOL;
    Load2 : BOOL;
    HMI_Int8 : INT;
    Warning_Cargo_NOK : BOOL;  (* Lift action with invalid cargo *)
    TCPReady : BOOL;
    RequestDriveReady : BOOL;
    DriveType : UINT;  (* 0=none, 1=docking, 2=buffer lane, 3=generic *)
    Lift_Height_Raw : INT;
    Navitrol_DistanceInfo : Navitrol_Status_DistanceToTarget_sec_struct;
    MES_Height_Req : UINT;  (* Desired height from MES *)
    Navitrol_FromTo : Navitrol_Status_FromTo_Sec_struct;
    Indicator_Left : BOOL;
    Indicator_Right : BOOL;
    K11 : BOOL;
    K12 : BOOL;
    Lift_Control_Dir : BOOL;
    Load_Distance : INT;
    HMI_Manual : BOOL;
    HMI_Int10 : INT;
    HMI_MessageCount : INT;
    SafetyStopped : BOOL;
    AgvLoaded : BOOL;  (* Object loaded *)
    Scanner1_State : State_Scanner;
    Scanner2_State : State_Scanner;
    Scanner3_State : State_Scanner;
    HMI_Input9 : BOOL;
    ClientConnected : BOOL;
    MES_Target : MQTT_Actuator_Request_struct;
    ENC1_Position : DINT;
    Navitrol_ProductionStatus : Navitrol_ProductionData_struct;
    RequestProductionStatus : BOOL;
    Navitrol_ProdDataStatusResult : UINT;
    HMI_Unload : BOOL;
    MES_Request_Cancel : BOOL;  (* Operator requests cancel for action *)
    Warning_Mqtt_Client_Error : BOOL;
    Mqtt_values : ARRAY[0..32] OF MQTTval;
    MQTT_enabled : BOOL;
    SafetyFieldNumber : INT;
    Pressure_Sensor_Load : BOOL;
    Scan1_Warn : BOOL;
    Scan3_Warn : BOOL;
    Scan1_Slow : BOOL;
    Scan3_slow : BOOL;
    Scan1_Stop : BOOL;
    Scan2_Stop : BOOL;
    MES_PalletDetection : Palletdetection_Action;
    CountedPallets : INT;
    PalletDetection_state : Pallet_Det_State;
    lift_heavyLoad : BOOL;
    RS232_OverhangDetected : BOOL;
    Lift_Controller_Error : BOOL;
    Scan2_Warn : BOOL;  (* Front left waring field *)
    Scan2_Slow : BOOL;  (* Front left stop field *)
    Scan3_Stop : BOOL;
    Lift_Sensor_Max : BOOL;
    Navitrol_Cust : Navitrol_Status_Custom_sec_struct;
    todo : BOOL;
    Dir_AGV : BOOL;  (* 0 = Forward *)
    AGV_Docking_Lane : BOOL;
    RequestTargetDetectionStatusV2 : BOOL;
    Navitrol_TargetDetectionStatus : Navitrol_TargetDetectionStatus_struct;
    Navitrol_TargetDetectionStatusToMES : Navitrol_TargetDetectionStatusToMes_struct;
    Navitrol_ErrorWithLevel : Navitrol_ErrorWithLevel_Struct;
    MaxSteeringAngleLaneDropping : REAL;
    AGVusesLowObstDetect : BOOL;
    LowObstacleIO : BOOL;
    MES_Popup : MQTT_Popup_struct;
    HMI_Input11 : BOOL;
    HMI_Input12 : BOOL;
    HMI_Int11 : INT;
    HMI_String1 : STRING[128];
    Manual_Mode : BOOL;
    O_LED_R : BOOL;
    O_LED_G : BOOL;
    O_LED_B : BOOL;
    MES_Language : INT;
    HMI_Int16 : INT;
    BufferLaneNavitrol_speed_limiter : BOOL;
    eLaneStateMES : Lane_state_MES;
    AGV_Lane : BOOL;
    AGV_LaneDocking : BOOL;
    AGV_LaneField : BOOL;
    HMI_Output8 : BOOL;
    HMI_Output12 : BOOL;
    BufferLaneSensorDistance : INT;
    Clamp : stClamp;
    NearTarget_No_Load : bool;
END_VAR
VAR
    _e1 : R_TRIG;
    _e2 : R_TRIG;
    _e3 : R_TRIG;
    _e4 : R_TRIG;
    _e5 : R_TRIG;
    _e6 : F_TRIG;
    _p7 : BOOL;
    _e8 : F_TRIG;
    _e9 : R_TRIG;
    _e10 : R_TRIG;
    _e11 : R_TRIG;
    _p12 : BOOL;
    _e13 : R_TRIG;
    _p14 : BOOL;
    _e15 : R_TRIG;
    _p16 : BOOL;
    _p17 : BOOL;
    _p18 : BOOL;
    _p19 : BOOL;
    _e20 : R_TRIG;
    _e21 : F_TRIG;
    _p22 : BOOL;
    _e23 : R_TRIG;
    _e24 : F_TRIG;
    _p25 : BOOL;
    _e26 : F_TRIG;
    _e27 : F_TRIG;
    _e28 : R_TRIG;
    _e29 : F_TRIG;
    _e30 : R_TRIG;
    _e31 : R_TRIG;
    _e32 : R_TRIG;
    _e33 : R_TRIG;
    _e34 : R_TRIG;
    _e35 : R_TRIG;
    _e36 : R_TRIG;
    _p37 : BOOL;
    _br75_0 : BOOL;
    _br75_1 : BOOL;
    _br75_2 : BOOL;
    _br76_0 : BOOL;
    _br76_1 : BOOL;
    _br76_2 : BOOL;
    _e38 : R_TRIG;
    _e39 : F_TRIG;
    _e40 : R_TRIG;
    _e41 : R_TRIG;
    _e42 : R_TRIG;
    _e43 : F_TRIG;
    _e44 : R_TRIG;
    _e45 : F_TRIG;
    _e46 : F_TRIG;
    _e47 : R_TRIG;
    _p48 : BOOL;
    _e49 : R_TRIG;
    _e50 : R_TRIG;
END_VAR

(* Section General: ladder, written here as Structured Text *)

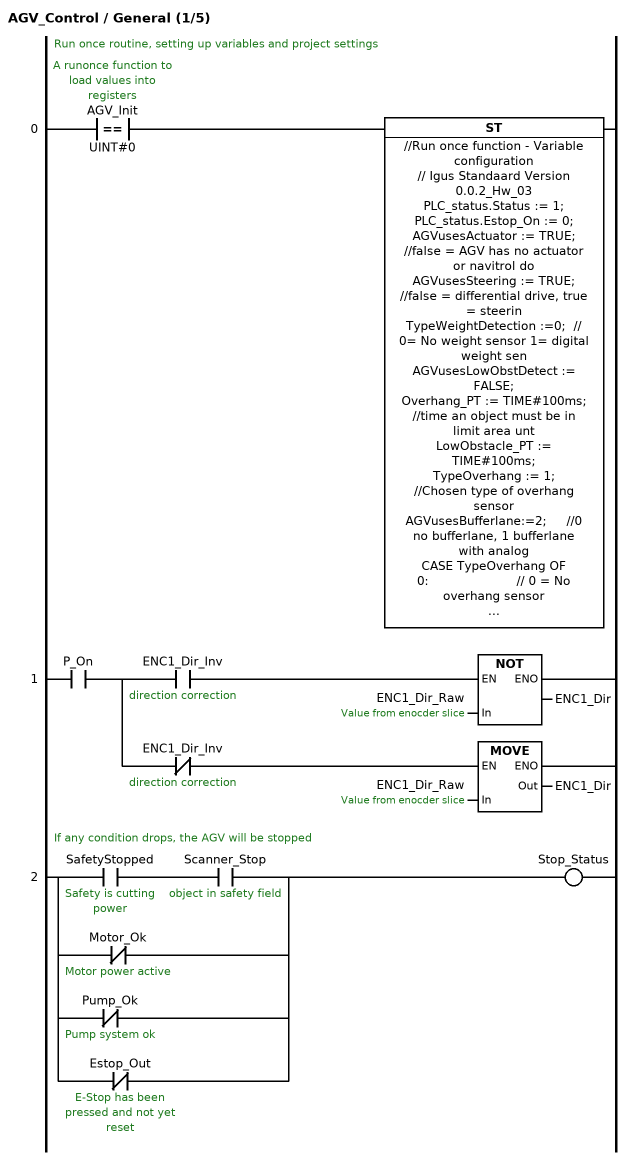
(* Rung 0: Run once routine, setting up variables and project settings *)
IF AGV_Init = UINT#0 THEN
    //Run once function - Variable configuration
    // Igus Standaard Version  0.0.2_Hw_03
    
    
    PLC_status.Status := 1;
    PLC_status.Estop_On := 0;
    AGVusesActuator := TRUE;	//false = AGV has no actuator or navitrol does not control it
    AGVusesSteering := TRUE;	//false = differential drive, true = steering wheel
    TypeWeightDetection :=0;  // 0= No weight sensor 1= digital weight sensor 2= analog weight sensor. 
    AGVusesLowObstDetect := FALSE;
    Overhang_PT := TIME#100ms;  //time an object must be in limit area until waring becomes active
    LowObstacle_PT := TIME#100ms; 
    TypeOverhang := 1;				//Chosen type of overhang sensor
    AGVusesBufferlane:=2;			//0 no bufferlane, 1 bufferlane with analog sensor, 2 bufferlane with scanners
    CASE TypeOverhang OF 
    0:											// 0 = No overhang sensor
    AGVusesRS232 := FALSE;		
    AGVusesSickOverhang := FALSE;
    1:											// 1 = RS232 overhang Lidar sensor (PF)
    AGVusesRS232 := TRUE;
    AGVusesSickOverhang := FALSE;
    2:											// 2 = I/O overhang sensor (SICK)
    AGVusesRS232 := FALSE;
    AGVusesSickOverhang := TRUE;
    END_CASE;
    
    mPerRot := 0.722;				//Distance traveled in m per wheel rotation
    WheelEncPpr := 29593.6;			//Encoder pulses per wheel roatation (PPR * gear ratio)
    UnloadDistance := 2000;	//Travel distance after unloading to clear load (or auto-reset lift)
    Max_docking_length := 200;	//Maximum travel distance when in docking in buffer lanes
    SilentMode :=FALSE;			//true = AGV starts in silent ControlModeLift
    AGVhasHandheld := FALSE;	//true = AGV has a remote control fixed to the AGV
    AGV_HasDoors := TRUE;		//true = AGV can be stopped if covers are open
    AnalogLoad := TRUE;			//true = AGV uses an analog sensor to detect objects over fork
    IF (AnalogLoad) THEN
    	AnalogLoad_Max := 1360;	//value when the sensor detects an object on the fork
    	AnalogLoad_Min := -60;		//minimal permitted value for load
    	AnalogLoad_Cargo_Max := 140;	//range where a load is far enough on the forks (must be higher than AnalogLoad_Min)
    END_IF;
    AGV_MaxSpeed := 1.6;		//AGV max speed in m/s
    AGV_DockingSpeed := 0.2;	//AGV docking speed in m/s
    NavitrolArrayLimit := FALSE;	//use speed array message to limit navitrol speed
    NavitrolSpeedLimit := TRUE;	//use speed limit message to limit navitrol speed
    NavitrolCommunication := TRUE;	//true = AGV can use navitrol communication
    NavithorCommunication := FALSE;	//true = AGV can communicate directly with navithor
    MQTT_enabled := TRUE;			//AGV usues MQTT communication with MES
    FINS_enabled := FALSE;			//AGV uses FINS communication with MES
    
    Scanner_WireReset_Enable := TRUE;	//Reset for Leuze available
    DomeLEDS := FALSE; //When true -> bowl leds, otherwise stripleds
    
    //Lift settings
    LiftHeightEmpty := 300;				//Height in mm for empty fork
    LiftHeightLoaded := 300; 				//Height in mm for fork with cargo
    Lift_Height_Drop := 90;					//Height in mm for drop/pick from floor
    LiftHeightMin := 88;						//Minimal value (in mm from floor) that can be used by fork
    LiftHeightMax:= 1280;	        		//Maximal value empty pallet (in mm from floor) that can be used by fork
    Lift_Height_Docking := 280; 			//Height in mm below which the lift should request docking
    LiftLimitMin:= 87;
    LiftLimitMax:=1285;
    LiftHeightHeavyLoadMax := 300; // Maximum height with heavy load
    
    //other settings
    LED_Ramp_Offset := 113;		//Ramp brightness where LEDs start to damp from (40 for low res, 113 for high res)
    LED_Ramp_Period := TIME#1s;	//Time when LEDs will fade
    
    CASE (MachineID) OF
    	11: 
    		LiftHeightScale := 0.15628;
    		LiftHeightOffset := -22;//-155;
    		Load_Distance_Scale:=0.174729;
    		Load_Distance_Offset:=2;
    		ENC1_Dir_Inv := TRUE;
    	12:
    		LiftHeightScale := 0.156519;
    		LiftHeightOffset := -30;
    		Load_Distance_Scale:=0.165201 ;
    		Load_Distance_Offset:=2;
    		ENC1_Dir_Inv := TRUE;
    	13: 
    		LiftHeightScale := 0.31292;
    		LiftHeightOffset := -216;
    		Load_Distance_Scale:=0.236292 ;
    		Load_Distance_Offset:=22;
    		ENC1_Dir_Inv := TRUE;
    	14: 
    		LiftHeightScale := 0.31292;
    		LiftHeightOffset := -216;
    		Load_Distance_Scale:=0.236292 ;
    		Load_Distance_Offset:=22;
    		ENC1_Dir_Inv := TRUE;
    	15: 
    		LiftHeightScale := 0.31292;
    		LiftHeightOffset := -216;
    		Load_Distance_Scale:=0.236292 ;
    		Load_Distance_Offset:=22;
    		ENC1_Dir_Inv := TRUE;
    	16: 
    		LiftHeightScale := 0.31292;
    		LiftHeightOffset := -216;
    		Load_Distance_Scale:=0.236292 ;
    		Load_Distance_Offset:=22;
    		ENC1_Dir_Inv := TRUE;
    ELSE
    	//optional default values
    	Lift_Height_Scale := 1;
    	Lift_Height_Offset := 0;
    	ENC1_Dir_Inv := FALSE;
    END_CASE;
    
    //Navitrol TCP configuration setup
    Navitrol_IP := '192.168.127.1';
    Navitrol_TX_Port:=5015;
    Navitrol_RX_Port:=0;
    
    //Navitrol tags
    DockingTag := 50;		//virtual tag ID to enable docking ControlModeLift
    NoDockingTag := 51;	//virtual tag ID to disable docking ControlModeLift (speed > 0.25 m/s will also disable docking)
    ChargerTag := 55;		//virtual tag ID to indicate a charger (result is AGV dependent)
    ToChargerTag := 56;	//virtual tag ID that disables overhang sensor so the AGV can reach the charger
    Tag_LaneField := 60; //Enable lanefield.
    Tag_DockingLaneField := 61; //Enable docking lanefield.
    
    //PLC -> Navitrol status section list
    //Section 1 is set/cleared with "AGVusesActuator"
    Navitrol_ManualSection_Enabled := FALSE;	//True if PLC is using navitrol's manual control
    Navitrol_ErrorSection_Enabled := FALSE;			//True if PLC sends errors and warnings to navitrol
    Navitrol_InputSection_Enabled := FALSE;		//True if PLC sends custom data to MES
    Navitrol_LaserSection_Enabled := TRUE;			//True if PLC controls more waning/stop fields than navitrol can handle (includes non-safe scanners and sensors)
    
    //Navitrol -> PLC status section list
    RequestGeneralSection := TRUE;						//general section should always be requested
    RequestHoldSection := FALSE;						//request hold section, can be used if AGV is allowed to release itself from hold-points
    RequestVirtualTagSection := TRUE;					//request information on virtual tags in the route (used for docking ControlModeLift)
    RequestComingGoingSection := FALSE;			//request navithor information about drive orders
    RequestCustomAtributeSection := TRUE; 		//not yet implemented, do not set to true
    RequestWarningSection := FALSE;					//request information about warning fields monitored by navitrol
    RequestOutputsSection := FALSE;					//request MES custom data (output messages from MES -> navithor) 
    RequestBatterySection := TRUE;						//Request battery data from navitrol (BMI by navitrol)
    RequestDriveInfoSection := TRUE;				
    RequestDistanceInfoSection := TRUE;		
    
    //***********************
    // !NOTE! Maximum of 10 sections. 
    // Each AGVuses... variable on TRUE adds 1 section!
    //***********************
    
    //prepare requested section IDs
    NrOfSections := 0;
    IF (RequestGeneralSection) THEN
    	//section ID 1, general
    	NrOfSections := NrOfSections +1;
    	Sections[1] := 1;
    	//general section is allways requested
    END_IF;
    
    IF (RequestHoldSection) THEN
    	//section ID 2, hold
    	NrOfSections := NrOfSections +1;
    	FOR index:=1 TO INT#10 DO
    		IF Sections[index] = 0 THEN
    			Sections[index] := 2;	//enter section ID
    			EXIT;								//section added to array, leave for loop
    		END_IF;
    	END_FOR;
    END_IF;
    
    IF (RequestVirtualTagSection) THEN
    	//section ID 3, virtual tag
    	NrOfSections := NrOfSections +1;
    	FOR index:=1 TO INT#10 DO
    		IF Sections[index] = 0 THEN
    			Sections[index] := 3;	//enter section ID
    			EXIT;								//section added to array, leave for loop
    		END_IF;
    	END_FOR;
    END_IF;
    
    IF (RequestComingGoingSection) THEN
    	//section ID 4, coming from & going to
    	NrOfSections := NrOfSections +1;
    	FOR index:=1 TO INT#10 DO
    		IF Sections[index] = 0 THEN
    			Sections[index] := 4;	//enter section ID
    			EXIT;								//section added to array, leave for loop
    		END_IF;
    	END_FOR;
    END_IF;
    
    IF (AGVusesActuator) THEN
    	//section ID 5, actuator
    	NrOfSections := NrOfSections +1;
    	FOR index:=1 TO INT#10 DO
    		IF Sections[index] = 0 THEN
    			Sections[index] := 5;	//enter section ID
    			EXIT;								//section added to array, leave for loop
    		END_IF;
    	END_FOR;
    	
    	//Actuator also needs to send data
    	Navitrol_ActSection_Enabled:= TRUE; //send actuator section
    	PLC_act.Section_ID := 1;
    	PLC_act.Section_Length := 14;
    	PLC_act.B_Inp.Load_Sensor_In_Use := 0;
    	IF (AgvLoaded) THEN
    		PLC_act.B_Inp.Load_Detected := 1;
    	ELSE
    		PLC_act.B_Inp.Load_Detected := 0;
    	END_IF;
    	PLC_act.B_Inp.Reserved_1 := 0;
    	PLC_act.B_Inp.Reserved_2 := 0;
    	PLC_act.B_Inp.Reserved_3 := 0;
    	PLC_act.B_Inp.Binary_Inputs_2 := 0;
    	PLC_act.B_Inp.Binary_Inputs_3 := 0;
    	PLC_act.B_Inp.Binary_Inputs_4 := 0;
    	
    	//check if lift is allready at bottom/top
    	IF (Lift_Bot_Pos=0 & Lift_Top_Pos=1) THEN PLC_act.Actr_Val := 0;
    	ELSIF (Lift_Bot_Pos=1 & Lift_Top_Pos=0) THEN PLC_act.Actr_Val := 2;
    	ELSE PLC_act.Actr_Val := 1;
    	END_IF;
    	
    	//the vehicle has an actuator, so that section is added to the status
    	MessageLength := MessageLength + PLC_act.Section_Length;
    END_IF;
    
    IF (RequestCustomAtributeSection) THEN
    	//section ID 6, custom atribute section
    	NrOfSections := NrOfSections +1;
    	FOR index:=1 TO INT#10 DO
    		IF Sections[index] = 0 THEN
    			Sections[index] := 6;	//enter section ID
    			EXIT;								//section added to array, leave for loop
    		END_IF;
    	END_FOR;
    END_IF;
    
    IF (RequestWarningSection) THEN
    	//section ID 7, warning zone
    	NrOfSections := NrOfSections +1;
    	FOR index:=1 TO INT#10 DO
    		IF Sections[index] = 0 THEN
    			Sections[index] := 7;	//enter section ID
    			EXIT;								//section added to array, leave for loop
    		END_IF;
    	END_FOR;
    END_IF;
    
    IF (RequestOutputsSection) THEN
    	//section ID 8, MES -> PLC outputs
    	NrOfSections := NrOfSections +1;
    	FOR index:=1 TO INT#10 DO
    		IF Sections[index] = 0 THEN
    			Sections[index] := 8;	//enter section ID
    			EXIT;								//section added to array, leave for loop
    		END_IF;
    	END_FOR;	
    END_IF;
    
    IF (AGVusesSteering) THEN
    	RequestSteeringAngleSection := TRUE;
    	//section ID 9, steering angle
    	NrOfSections := NrOfSections +1;
    	FOR index:=1 TO INT#10 DO
    		IF Sections[index] = 0 THEN
    			Sections[index] := 9;	//enter section ID
    			EXIT;								//section added to array, leave for loop
    		END_IF;
    	END_FOR;
    END_IF;
    
    IF (RequestBatterySection) THEN
    	//section ID 10, battery section
    	NrOfSections := NrOfSections +1;
    	FOR index:=1 TO INT#10 DO
    		IF Sections[index] = 0 THEN
    			Sections[index] := 10;	//enter section ID
    			EXIT;								//section added to array, leave for loop
    		END_IF;
    	END_FOR;
    END_IF;
    
    IF (RequestDriveInfoSection) THEN
    	//section ID 12, driveinfo section
    	NrOfSections := NrOfSections +1;
    	FOR index:=1 TO INT#10 DO
    		IF Sections[index] = 0 THEN
    			Sections[index] := 12;	//enter section ID
    			EXIT;								//section added to array, leave for loop
    		END_IF;
    	END_FOR;
    END_IF;
    
    IF (RequestDistanceInfoSection) THEN
    	//section ID 13, distanceinfo section
    	NrOfSections := NrOfSections +1;
    	FOR index:=1 TO INT#10 DO
    		IF Sections[index] = 0 THEN
    			Sections[index] := 13;	//enter section ID
    			EXIT;								//section added to array, leave for loop
    		END_IF;
    	END_FOR;
    END_IF;
    
    
    //run once, set AGV_init
    AGV_Init := 1;
END_IF;
(* Rung 1 *)
IF P_On AND ENC1_Dir_Inv THEN ENC1_Dir := NOT ENC1_Dir_Raw; END_IF;
IF P_On AND NOT ENC1_Dir_Inv THEN ENC1_Dir := ENC1_Dir_Raw; END_IF;
(* Rung 2: If any condition drops, the AGV will be stopped *)
Stop_Status := (SafetyStopped AND Scanner_Stop) OR NOT Motor_Ok OR NOT Pump_Ok OR NOT Estop_Out;

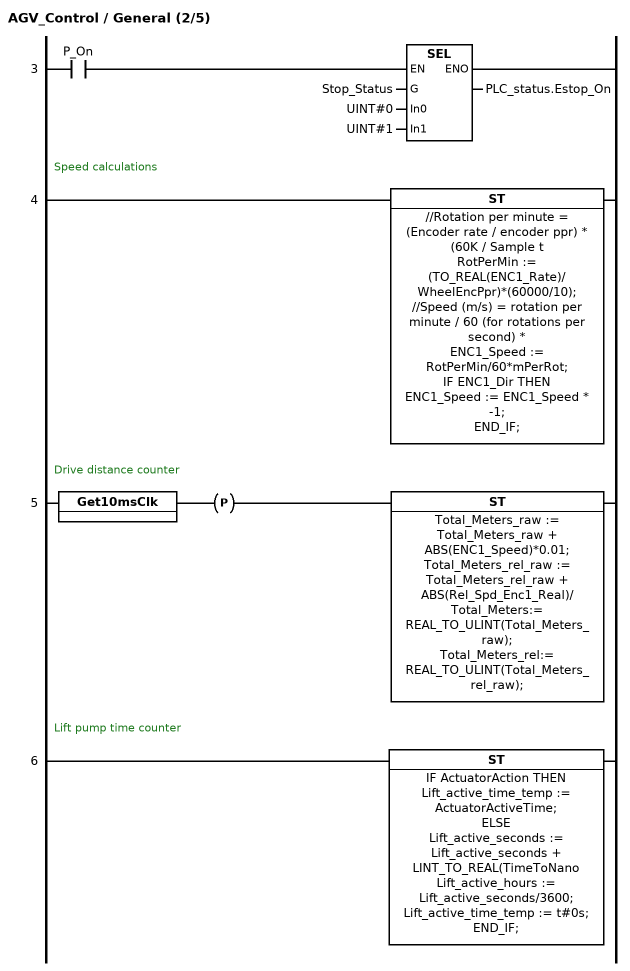
(* Rung 3 *)
IF P_On THEN PLC_status.Estop_On := SEL(G := Stop_Status, In0 := UINT#0, In1 := UINT#1); END_IF;
(* Rung 4: Speed calculations *)
//Rotation per minute = (Encoder rate / encoder ppr) * (60K / Sample time(in mSec))
RotPerMin := (TO_REAL(ENC1_Rate)/WheelEncPpr)*(60000/10);
//Speed (m/s) = rotation per minute / 60 (for rotations per second) * distance per rotation
ENC1_Speed := RotPerMin/60*mPerRot;
IF ENC1_Dir THEN
	ENC1_Speed := ENC1_Speed * -1;
END_IF;
(* Rung 5: Drive distance counter *)
_e1(CLK := Get10msClk());
IF _e1.Q THEN
    Total_Meters_raw := Total_Meters_raw + ABS(ENC1_Speed)*0.01;
    Total_Meters_rel_raw := Total_Meters_rel_raw + ABS(Rel_Spd_Enc1_Real)/100*0.01;
    Total_Meters:= REAL_TO_ULINT(Total_Meters_raw);
    Total_Meters_rel:= REAL_TO_ULINT(Total_Meters_rel_raw);
END_IF;
(* Rung 6: Lift pump time counter *)
IF ActuatorAction THEN
	Lift_active_time_temp := ActuatorActiveTime;
ELSE
	Lift_active_seconds := Lift_active_seconds + LINT_TO_REAL(TimeToNanoSec(Lift_active_time_temp))/1e9;
	Lift_active_hours := Lift_active_seconds/3600;
	Lift_active_time_temp := t#0s;
END_IF;

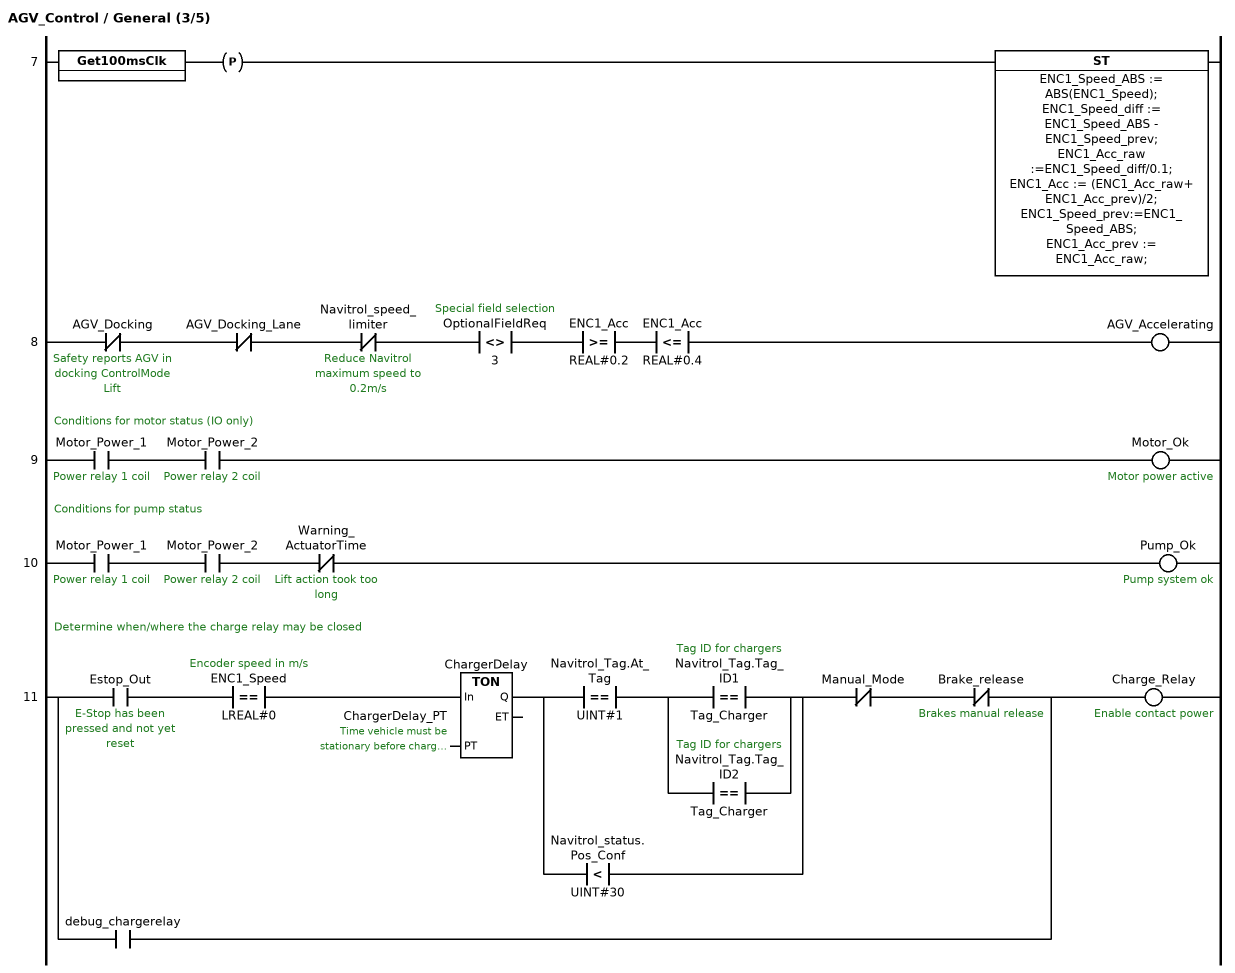
(* Rung 7 *)
_e2(CLK := Get100msClk());
IF _e2.Q THEN
    ENC1_Speed_ABS := ABS(ENC1_Speed);
    ENC1_Speed_diff := ENC1_Speed_ABS - ENC1_Speed_prev;
    ENC1_Acc_raw :=ENC1_Speed_diff/0.1;
    ENC1_Acc := (ENC1_Acc_raw+ ENC1_Acc_prev)/2;
    
    ENC1_Speed_prev:=ENC1_Speed_ABS;
    ENC1_Acc_prev := ENC1_Acc_raw;
END_IF;
(* Rung 8 *)
AGV_Accelerating := NOT AGV_Docking AND NOT AGV_Docking_Lane AND NOT Navitrol_speed_limiter AND (OptionalFieldReq <> 3) AND (ENC1_Acc >= REAL#0.2) AND (ENC1_Acc <= REAL#0.4);
(* Rung 9: Conditions for motor status (IO only) *)
Motor_Ok := Motor_Power_1 AND Motor_Power_2;
(* Rung 10: Conditions for pump status *)
Pump_Ok := Motor_Power_1 AND Motor_Power_2 AND NOT Warning_ActuatorTime;
(* Rung 11: Determine when/where the charge relay may be closed *)
ChargerDelay(In := Estop_Out AND (ENC1_Speed = LREAL#0), PT := ChargerDelay_PT);
Charge_Relay := (ChargerDelay.Q AND (((Navitrol_Tag.At_Tag = UINT#1) AND ((Navitrol_Tag.Tag_ID1 = Tag_Charger) OR (Navitrol_Tag.Tag_ID2 = Tag_Charger))) OR (Navitrol_status.Pos_Conf < UINT#30)) AND NOT Manual_Mode AND NOT Brake_release) OR debug_chargerelay;

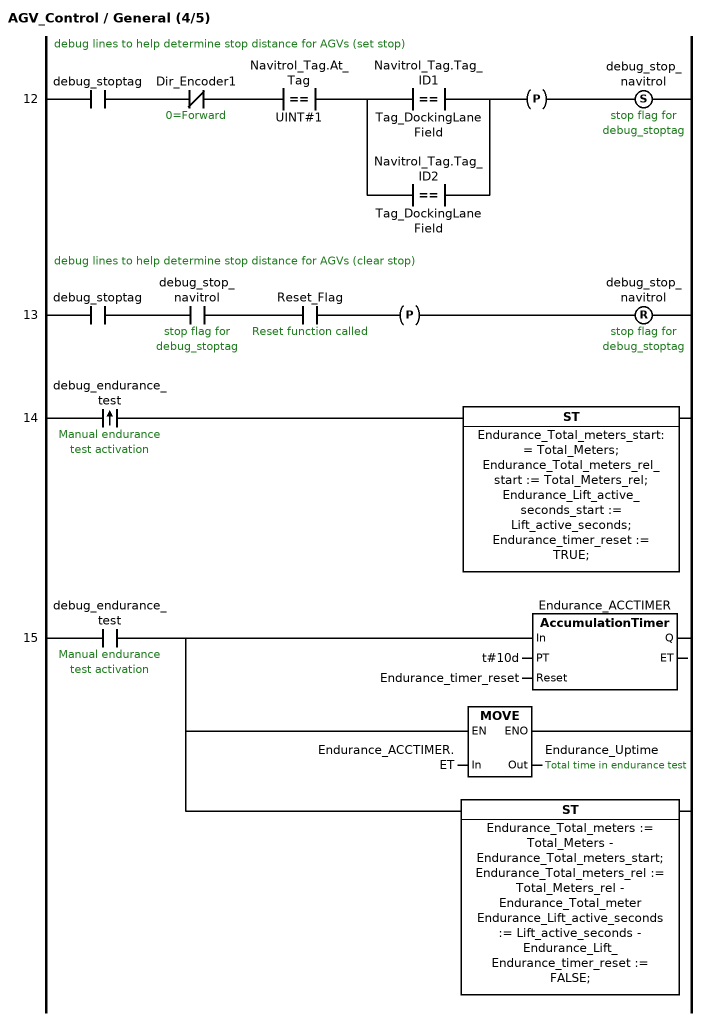
(* Rung 12: debug lines to help determine stop distance for AGVs (set stop) *)
_e3(CLK := debug_stoptag AND NOT Dir_Encoder1 AND (Navitrol_Tag.At_Tag = UINT#1) AND ((Navitrol_Tag.Tag_ID1 = Tag_DockingLaneField) OR (Navitrol_Tag.Tag_ID2 = Tag_DockingLaneField)));
IF _e3.Q THEN debug_stop_navitrol := TRUE; END_IF;
(* Rung 13: debug lines to help determine stop distance for AGVs (clear stop) *)
_e4(CLK := debug_stoptag AND debug_stop_navitrol AND Reset_Flag);
IF _e4.Q THEN debug_stop_navitrol := FALSE; END_IF;
(* Rung 14 *)
_e5(CLK := debug_endurance_test);
IF _e5.Q THEN
    Endurance_Total_meters_start:= Total_Meters;
    Endurance_Total_meters_rel_start := Total_Meters_rel;
    Endurance_Lift_active_seconds_start := Lift_active_seconds;
    Endurance_timer_reset := TRUE;
END_IF;
(* Rung 15 *)
Endurance_ACCTIMER(In := debug_endurance_test, PT := t#10d, Reset := Endurance_timer_reset);
IF debug_endurance_test THEN Endurance_Uptime := Endurance_ACCTIMER.ET; END_IF;
IF debug_endurance_test THEN
    Endurance_Total_meters := Total_Meters - Endurance_Total_meters_start;
    Endurance_Total_meters_rel := Total_Meters_rel - Endurance_Total_meters_rel_start;
    Endurance_Lift_active_seconds := Lift_active_seconds - Endurance_Lift_active_seconds_start;
    Endurance_timer_reset := FALSE;
END_IF;

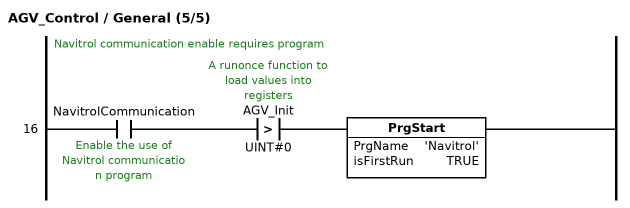
(* Rung 16: Navitrol communication enable requires program *)
(* drawn but driving nothing: NavitrolCommunication, AGV_Init, UINT#0, 'Navitrol', TRUE *)

(* Section Safety: ladder, written here as Structured Text *)

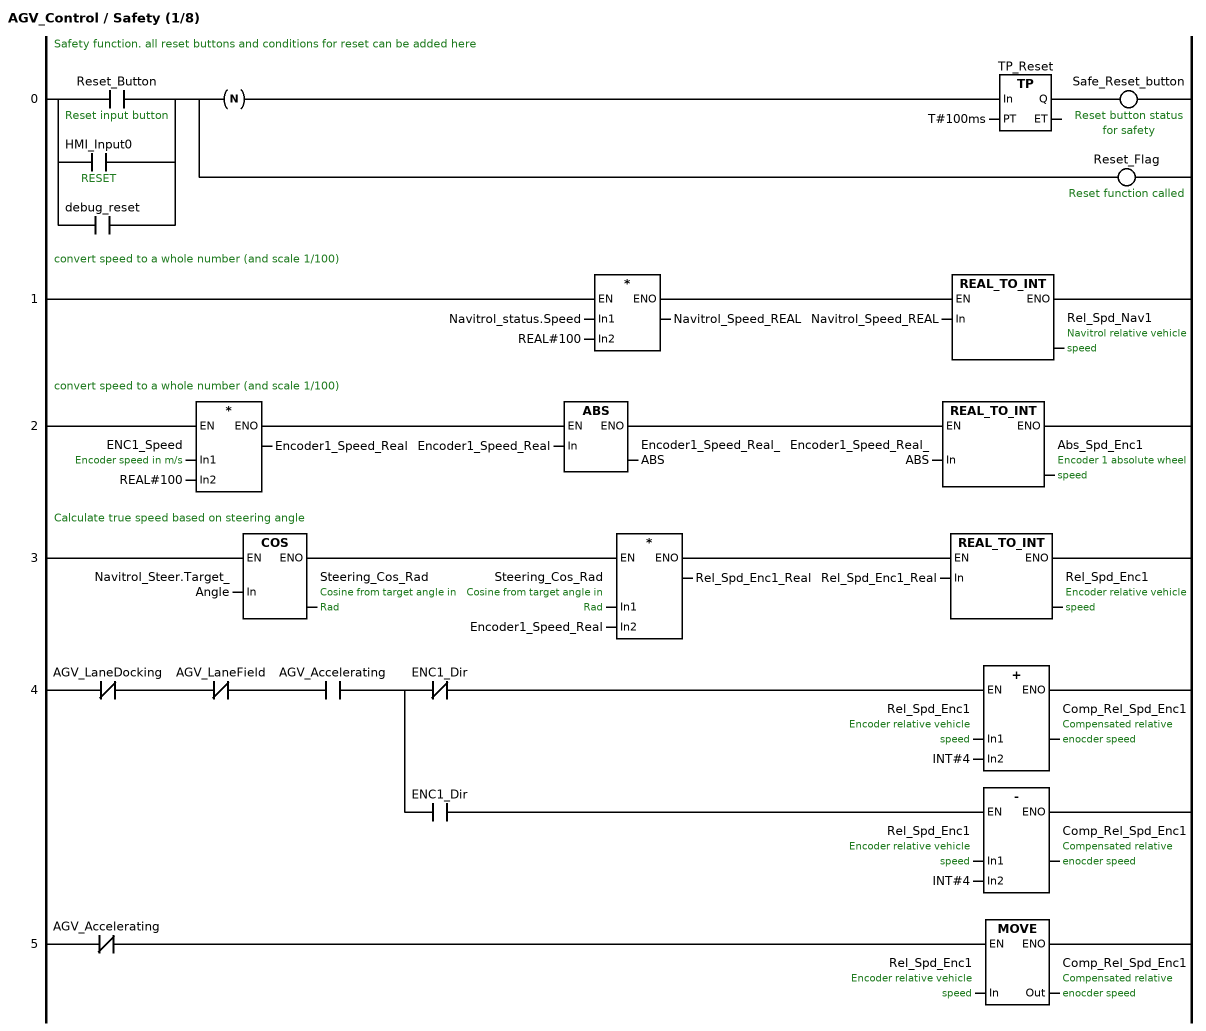
(* Rung 0: Safety function. all reset buttons and conditions for reset can be added here *)
_e6(CLK := Reset_Button OR HMI_Input0 OR debug_reset);
TP_Reset(In := _e6.Q, PT := T#100ms);
Safe_Reset_button := TP_Reset.Q;
Reset_Flag := Reset_Button OR HMI_Input0 OR debug_reset;
(* Rung 1: convert speed to a whole number (and scale 1/100) *)
Navitrol_Speed_REAL := Navitrol_status.Speed * REAL#100;
Rel_Spd_Nav1 := REAL_TO_INT(In := Navitrol_Speed_REAL);
(* Rung 2: convert speed to a whole number (and scale 1/100) *)
Encoder1_Speed_Real := ENC1_Speed * REAL#100;
Encoder1_Speed_Real_ABS := ABS(In := Encoder1_Speed_Real);
Abs_Spd_Enc1 := REAL_TO_INT(In := Encoder1_Speed_Real_ABS);
(* Rung 3: Calculate true speed based on steering angle *)
Steering_Cos_Rad := COS(In := Navitrol_Steer.Target_Angle);
Rel_Spd_Enc1_Real := Steering_Cos_Rad * Encoder1_Speed_Real;
Rel_Spd_Enc1 := REAL_TO_INT(In := Rel_Spd_Enc1_Real);
(* Rung 4 *)
_p7 := NOT AGV_LaneDocking AND NOT AGV_LaneField AND AGV_Accelerating;
IF _p7 AND NOT ENC1_Dir THEN Comp_Rel_Spd_Enc1 := Rel_Spd_Enc1 + INT#4; END_IF;
IF _p7 AND ENC1_Dir THEN Comp_Rel_Spd_Enc1 := Rel_Spd_Enc1 - INT#4; END_IF;
(* Rung 5 *)
IF NOT AGV_Accelerating THEN Comp_Rel_Spd_Enc1 := Rel_Spd_Enc1; END_IF;

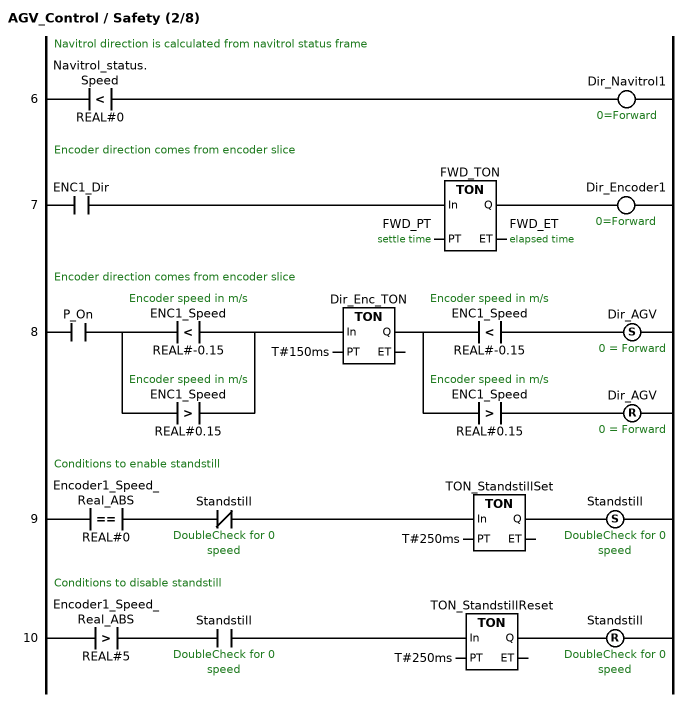
(* Rung 6: Navitrol direction is calculated from navitrol status frame *)
Dir_Navitrol1 := Navitrol_status.Speed < REAL#0;
(* Rung 7: Encoder direction comes from encoder slice *)
FWD_TON(In := ENC1_Dir, PT := FWD_PT, ET => FWD_ET);
Dir_Encoder1 := FWD_TON.Q;
(* Rung 8: Encoder direction comes from encoder slice *)
Dir_Enc_TON(In := P_On AND ((ENC1_Speed < (REAL#-0.15)) OR (ENC1_Speed > REAL#0.15)), PT := T#150ms);
IF Dir_Enc_TON.Q AND (ENC1_Speed < (REAL#-0.15)) THEN Dir_AGV := TRUE; END_IF;
IF Dir_Enc_TON.Q AND (ENC1_Speed > REAL#0.15) THEN Dir_AGV := FALSE; END_IF;
(* Rung 9: Conditions to enable standstill *)
TON_StandstillSet(In := (Encoder1_Speed_Real_ABS = REAL#0) AND NOT Standstill, PT := T#250ms);
IF TON_StandstillSet.Q THEN Standstill := TRUE; END_IF;
(* Rung 10: Conditions to disable standstill *)
TON_StandstillReset(In := (Encoder1_Speed_Real_ABS > REAL#5) AND Standstill, PT := T#250ms);
IF TON_StandstillReset.Q THEN Standstill := FALSE; END_IF;

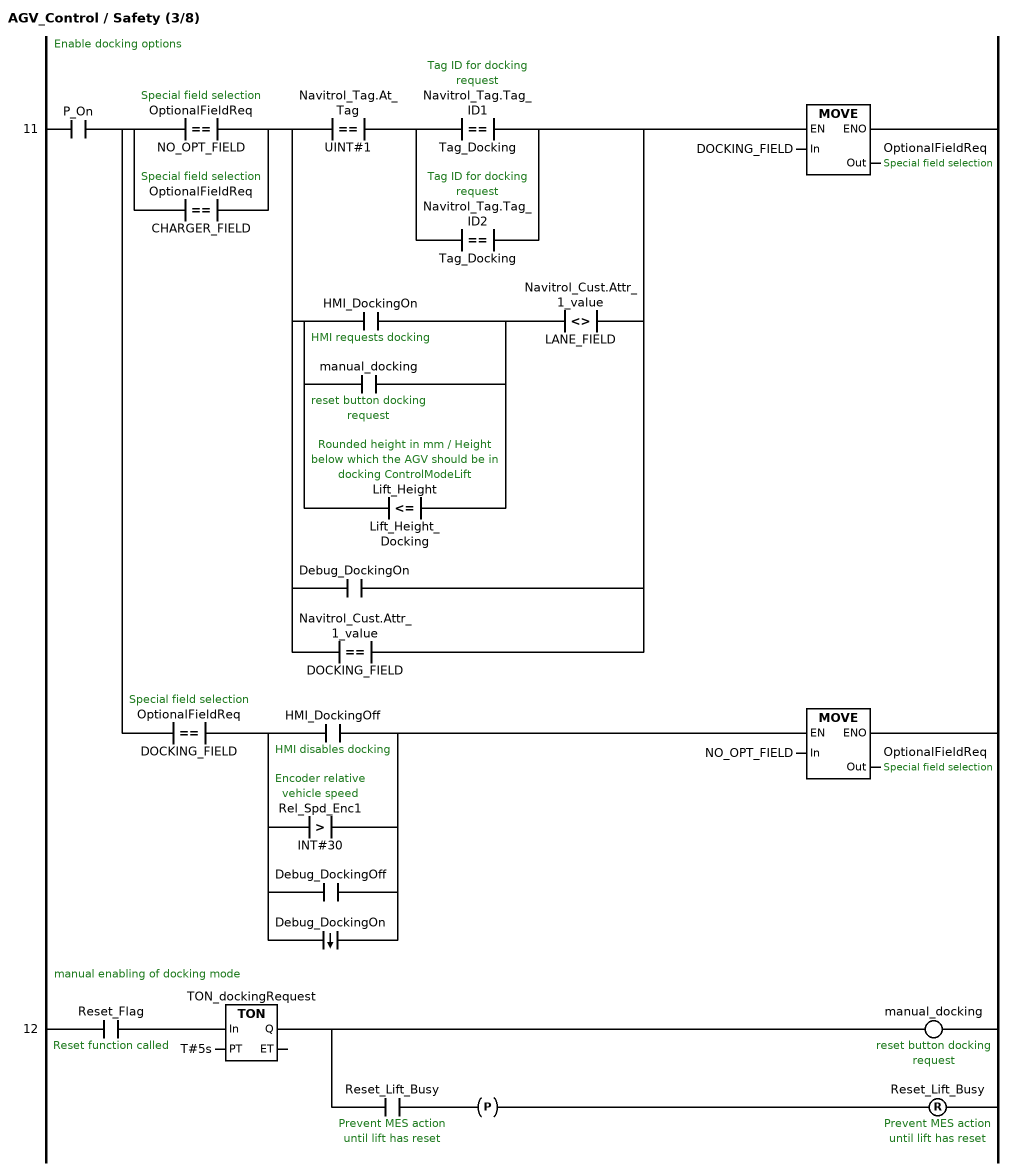
(* Rung 11: Enable docking options *)
IF P_On AND ((OptionalFieldReq = NO_OPT_FIELD) OR (OptionalFieldReq = CHARGER_FIELD)) AND (((Navitrol_Tag.At_Tag = UINT#1) AND ((Navitrol_Tag.Tag_ID1 = Tag_Docking) OR (Navitrol_Tag.Tag_ID2 = Tag_Docking))) OR ((HMI_DockingOn OR manual_docking OR (Lift_Height <= Lift_Height_Docking)) AND (Navitrol_Cust.Attr_1_value <> LANE_FIELD)) OR Debug_DockingOn OR (Navitrol_Cust.Attr_1_value = DOCKING_FIELD)) THEN
    OptionalFieldReq := DOCKING_FIELD;
END_IF;
_e8(CLK := Debug_DockingOn);
IF P_On AND (OptionalFieldReq = DOCKING_FIELD) AND (HMI_DockingOff OR (Rel_Spd_Enc1 > INT#30) OR Debug_DockingOff OR _e8.Q) THEN
    OptionalFieldReq := NO_OPT_FIELD;
END_IF;
(* Rung 12: manual enabling of docking mode *)
TON_dockingRequest(In := Reset_Flag, PT := T#5s);
manual_docking := TON_dockingRequest.Q;
_e9(CLK := TON_dockingRequest.Q AND Reset_Lift_Busy);
IF _e9.Q THEN Reset_Lift_Busy := FALSE; END_IF;

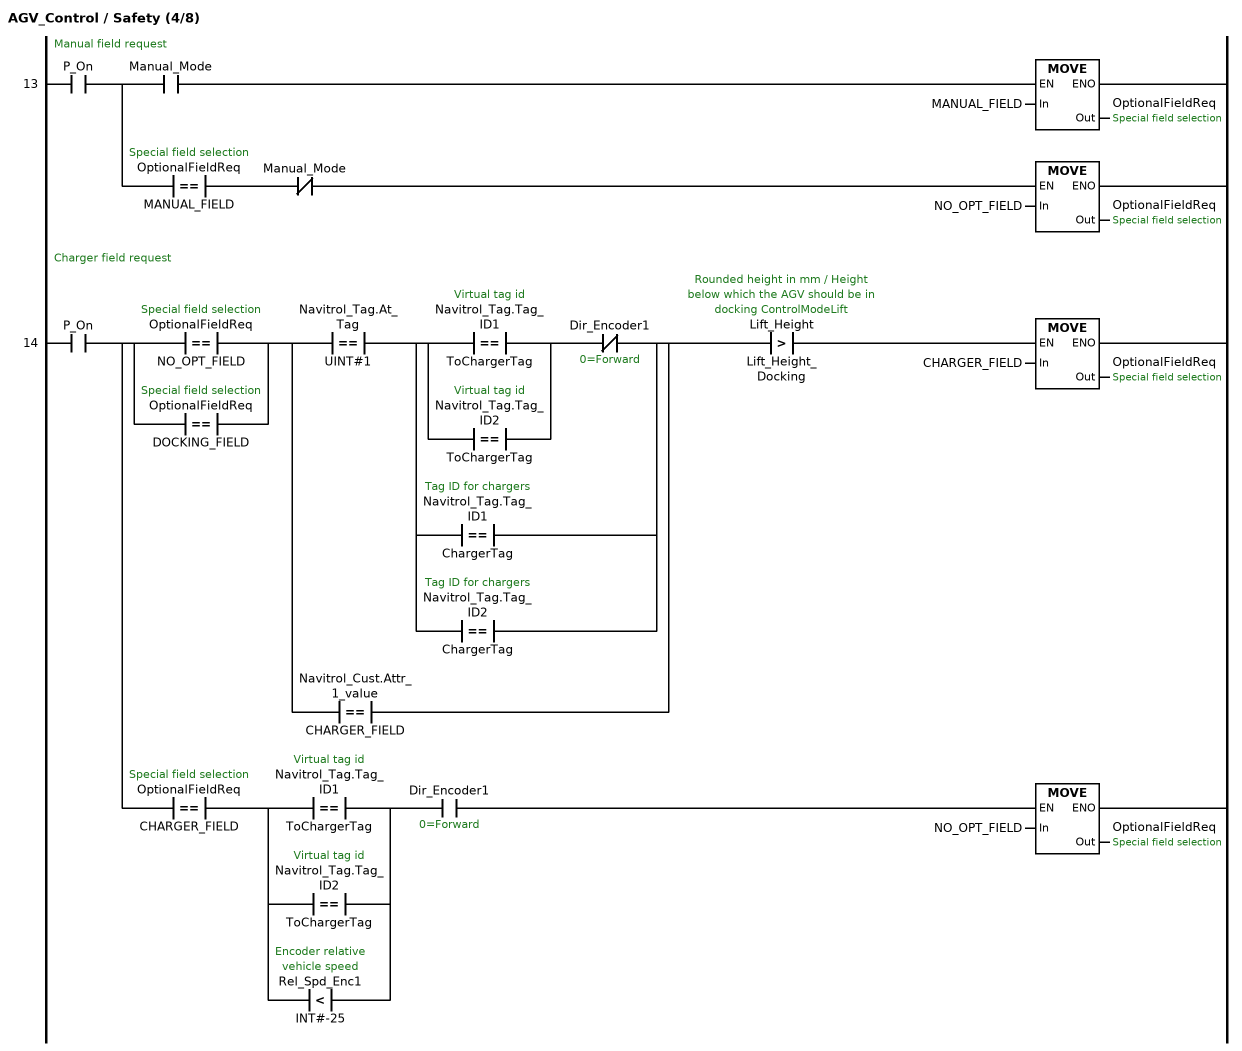
(* Rung 13: Manual field request *)
IF P_On AND Manual_Mode THEN OptionalFieldReq := MANUAL_FIELD; END_IF;
IF P_On AND (OptionalFieldReq = MANUAL_FIELD) AND NOT Manual_Mode THEN
    OptionalFieldReq := NO_OPT_FIELD;
END_IF;
(* Rung 14: Charger field request *)
IF P_On AND ((OptionalFieldReq = NO_OPT_FIELD) OR (OptionalFieldReq = DOCKING_FIELD)) AND (((Navitrol_Tag.At_Tag = UINT#1) AND ((((Navitrol_Tag.Tag_ID1 = ToChargerTag) OR (Navitrol_Tag.Tag_ID2 = ToChargerTag)) AND NOT Dir_Encoder1) OR (Navitrol_Tag.Tag_ID1 = ChargerTag) OR (Navitrol_Tag.Tag_ID2 = ChargerTag))) OR (Navitrol_Cust.Attr_1_value = CHARGER_FIELD)) AND (Lift_Height > Lift_Height_Docking) THEN
    OptionalFieldReq := CHARGER_FIELD;
END_IF;
IF P_On AND (OptionalFieldReq = CHARGER_FIELD) AND ((Navitrol_Tag.Tag_ID1 = ToChargerTag) OR (Navitrol_Tag.Tag_ID2 = ToChargerTag) OR (Rel_Spd_Enc1 < (INT#-25))) AND Dir_Encoder1 THEN
    OptionalFieldReq := NO_OPT_FIELD;
END_IF;

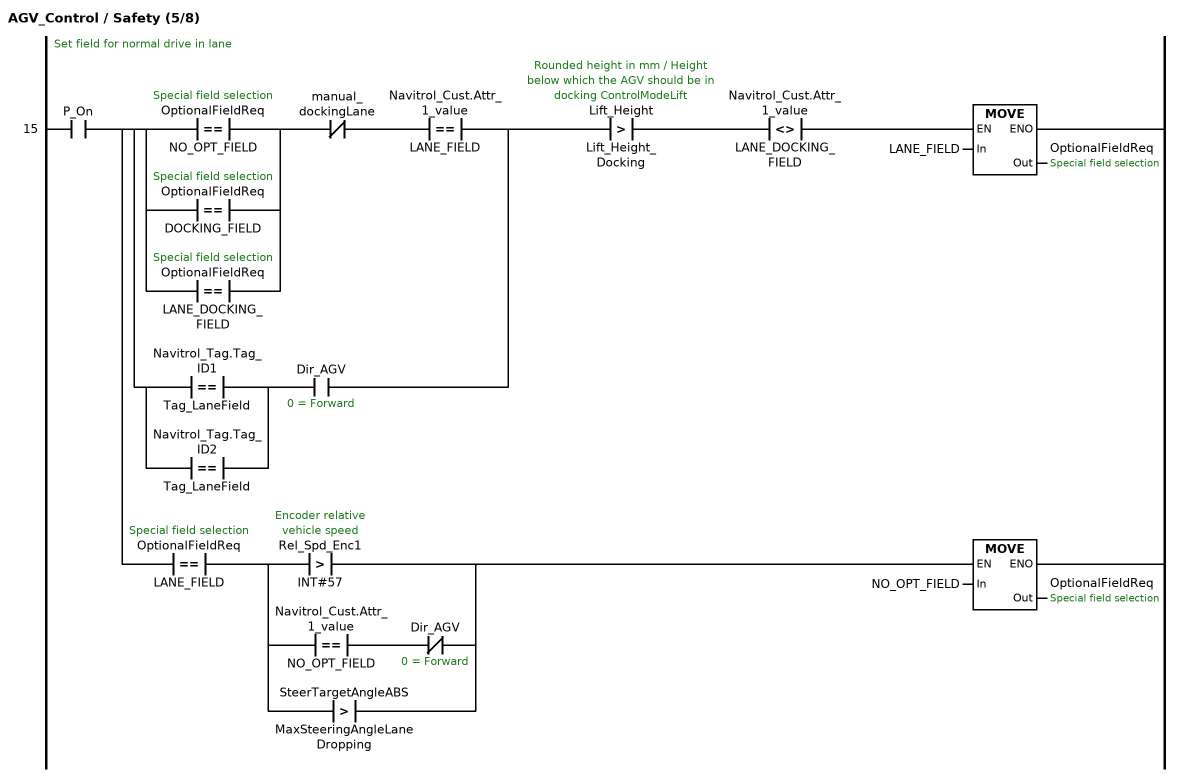
(* Rung 15: Set field for normal drive in lane *)
IF P_On AND ((((OptionalFieldReq = NO_OPT_FIELD) OR (OptionalFieldReq = DOCKING_FIELD) OR (OptionalFieldReq = LANE_DOCKING_FIELD)) AND NOT manual_dockingLane AND (Navitrol_Cust.Attr_1_value = LANE_FIELD)) OR (((Navitrol_Tag.Tag_ID1 = Tag_LaneField) OR (Navitrol_Tag.Tag_ID2 = Tag_LaneField)) AND Dir_AGV)) AND (Lift_Height > Lift_Height_Docking) AND (Navitrol_Cust.Attr_1_value <> LANE_DOCKING_FIELD) THEN
    OptionalFieldReq := LANE_FIELD;
END_IF;
IF P_On AND (OptionalFieldReq = LANE_FIELD) AND ((Rel_Spd_Enc1 > INT#57) OR ((Navitrol_Cust.Attr_1_value = NO_OPT_FIELD) AND NOT Dir_AGV) OR (SteerTargetAngleABS > MaxSteeringAngleLaneDropping)) THEN
    OptionalFieldReq := NO_OPT_FIELD;
END_IF;

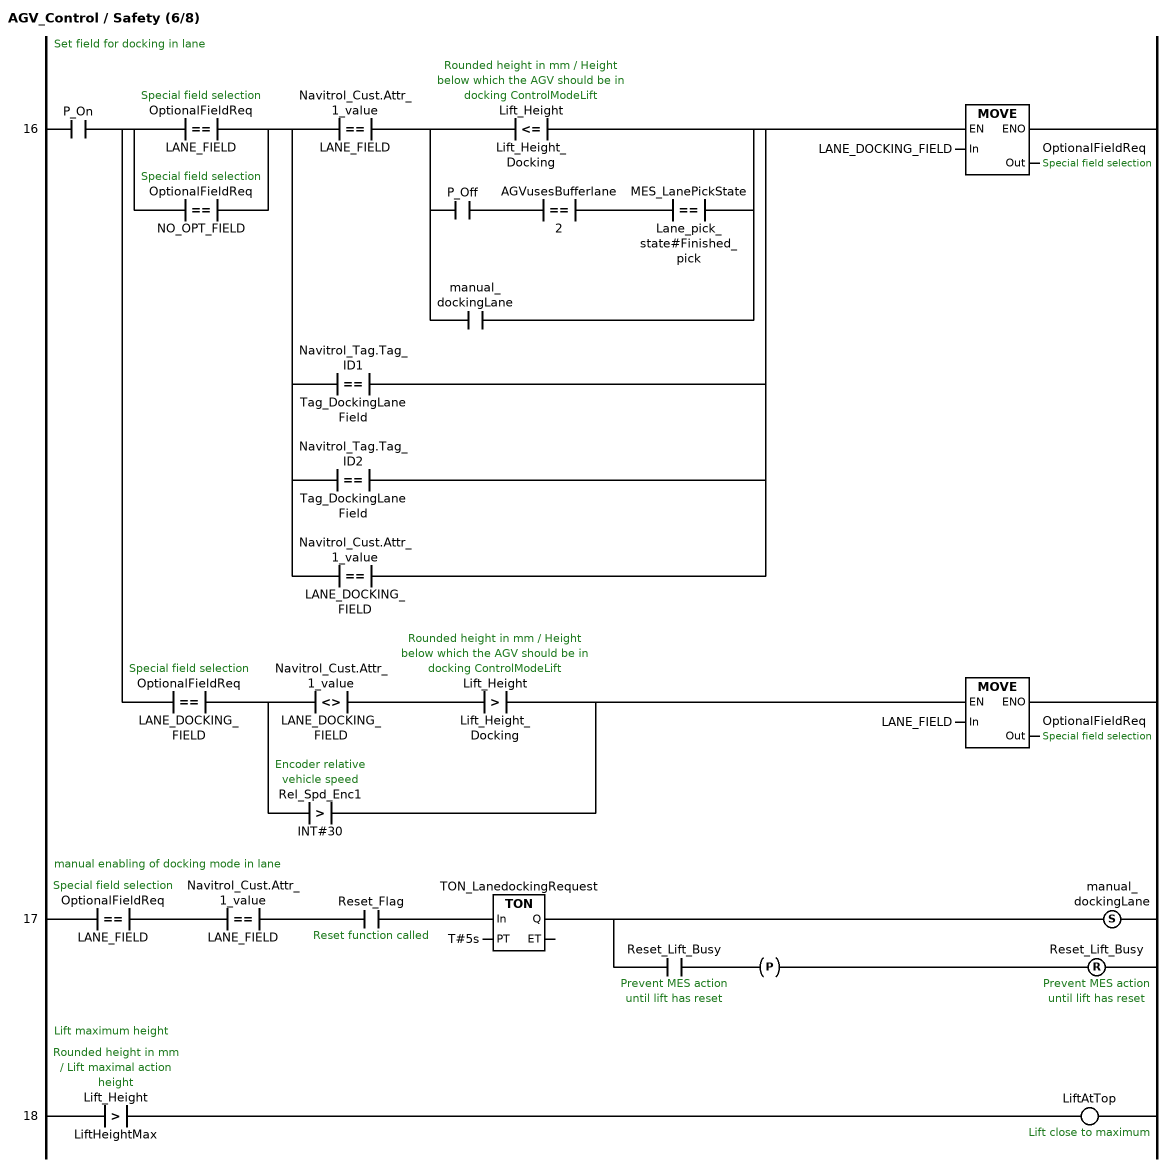
(* Rung 16: Set field for docking in lane *)
IF P_On AND ((OptionalFieldReq = LANE_FIELD) OR (OptionalFieldReq = NO_OPT_FIELD)) AND (((Navitrol_Cust.Attr_1_value = LANE_FIELD) AND ((Lift_Height <= Lift_Height_Docking) OR (P_Off AND (AGVusesBufferlane = 2) AND (MES_LanePickState = Lane_pick_state#Finished_pick)) OR manual_dockingLane)) OR (Navitrol_Tag.Tag_ID1 = Tag_DockingLaneField) OR (Navitrol_Tag.Tag_ID2 = Tag_DockingLaneField) OR (Navitrol_Cust.Attr_1_value = LANE_DOCKING_FIELD)) THEN
    OptionalFieldReq := LANE_DOCKING_FIELD;
END_IF;
IF P_On AND (OptionalFieldReq = LANE_DOCKING_FIELD) AND (((Navitrol_Cust.Attr_1_value <> LANE_DOCKING_FIELD) AND (Lift_Height > Lift_Height_Docking)) OR (Rel_Spd_Enc1 > INT#30)) THEN
    OptionalFieldReq := LANE_FIELD;
END_IF;
(* Rung 17: manual enabling of docking mode in lane *)
TON_LanedockingRequest(In := (OptionalFieldReq = LANE_FIELD) AND (Navitrol_Cust.Attr_1_value = LANE_FIELD) AND Reset_Flag, PT := T#5s);
IF TON_LanedockingRequest.Q THEN manual_dockingLane := TRUE; END_IF;
_e10(CLK := TON_LanedockingRequest.Q AND Reset_Lift_Busy);
IF _e10.Q THEN Reset_Lift_Busy := FALSE; END_IF;
(* Rung 18: Lift maximum height *)
LiftAtTop := Lift_Height > LiftHeightMax;

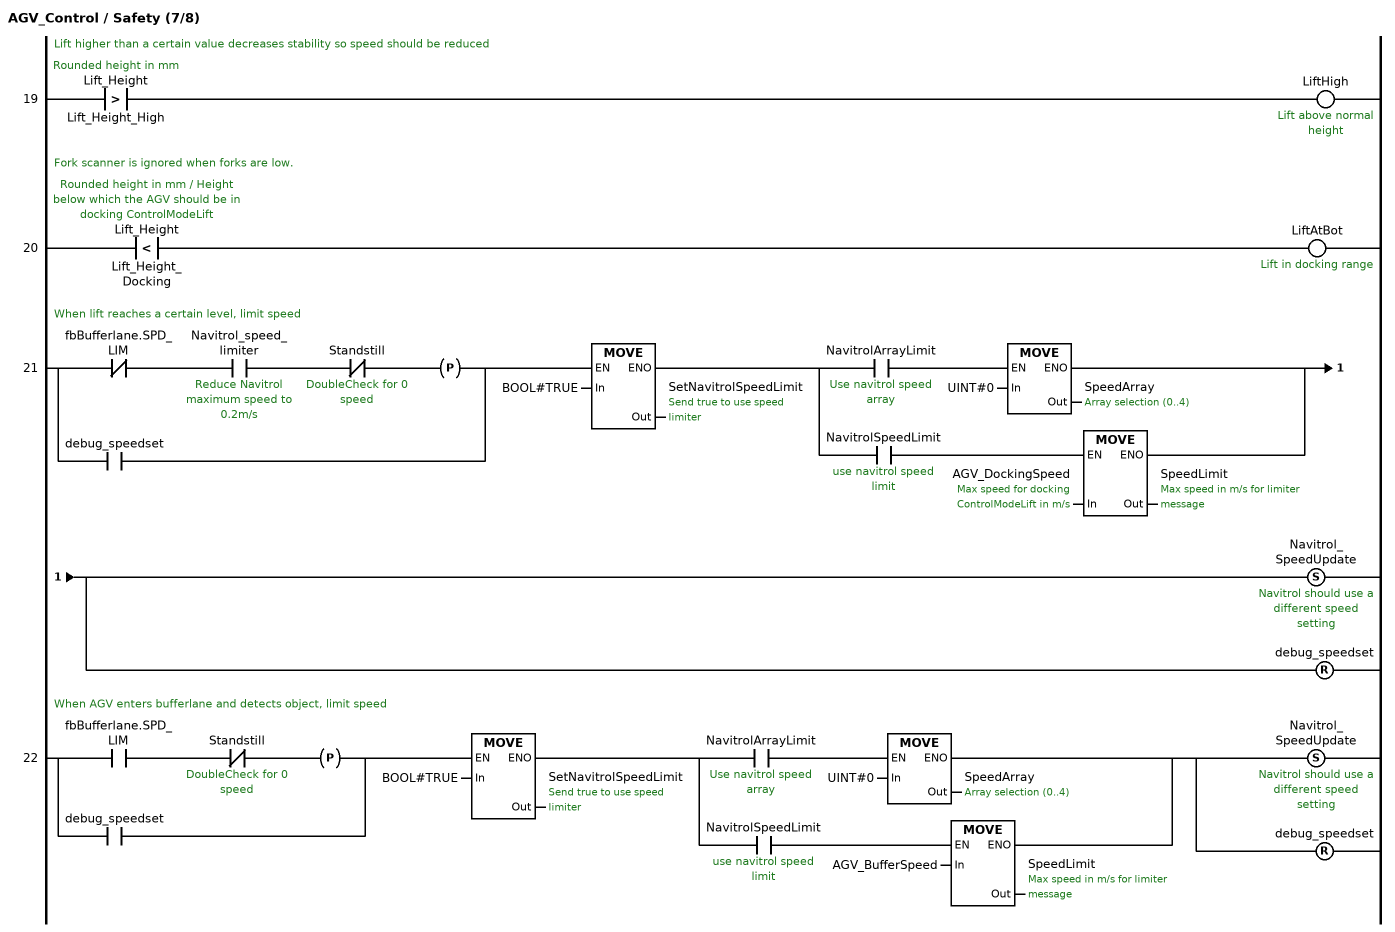
(* Rung 19: Lift higher than a certain value decreases stability so speed should be reduced *)
LiftHigh := Lift_Height > Lift_Height_High;
(* Rung 20: Fork scanner is ignored when forks are low. *)
LiftAtBot := Lift_Height < Lift_Height_Docking;
(* Rung 21: When lift reaches a certain level, limit speed *)
_e11(CLK := NOT fbBufferlane.SPD_LIM AND Navitrol_speed_limiter AND NOT Standstill);
IF _e11.Q OR debug_speedset THEN SetNavitrolSpeedLimit := BOOL#TRUE; END_IF;
IF (_e11.Q OR debug_speedset) AND NavitrolArrayLimit THEN SpeedArray := UINT#0; END_IF;
IF (_e11.Q OR debug_speedset) AND NavitrolSpeedLimit THEN SpeedLimit := AGV_DockingSpeed; END_IF;
_p12 := (_e11.Q OR debug_speedset) AND (NavitrolArrayLimit OR NavitrolSpeedLimit);
IF _p12 THEN
    Navitrol_SpeedUpdate := TRUE;
    debug_speedset := FALSE;
END_IF;
(* Rung 22: When AGV enters bufferlane and detects object, limit speed *)
_e13(CLK := fbBufferlane.SPD_LIM AND NOT Standstill);
IF _e13.Q OR debug_speedset THEN SetNavitrolSpeedLimit := BOOL#TRUE; END_IF;
IF (_e13.Q OR debug_speedset) AND NavitrolArrayLimit THEN SpeedArray := UINT#0; END_IF;
IF (_e13.Q OR debug_speedset) AND NavitrolSpeedLimit THEN SpeedLimit := AGV_BufferSpeed; END_IF;
_p14 := (_e13.Q OR debug_speedset) AND (NavitrolArrayLimit OR NavitrolSpeedLimit);
IF _p14 THEN
    Navitrol_SpeedUpdate := TRUE;
    debug_speedset := FALSE;
END_IF;

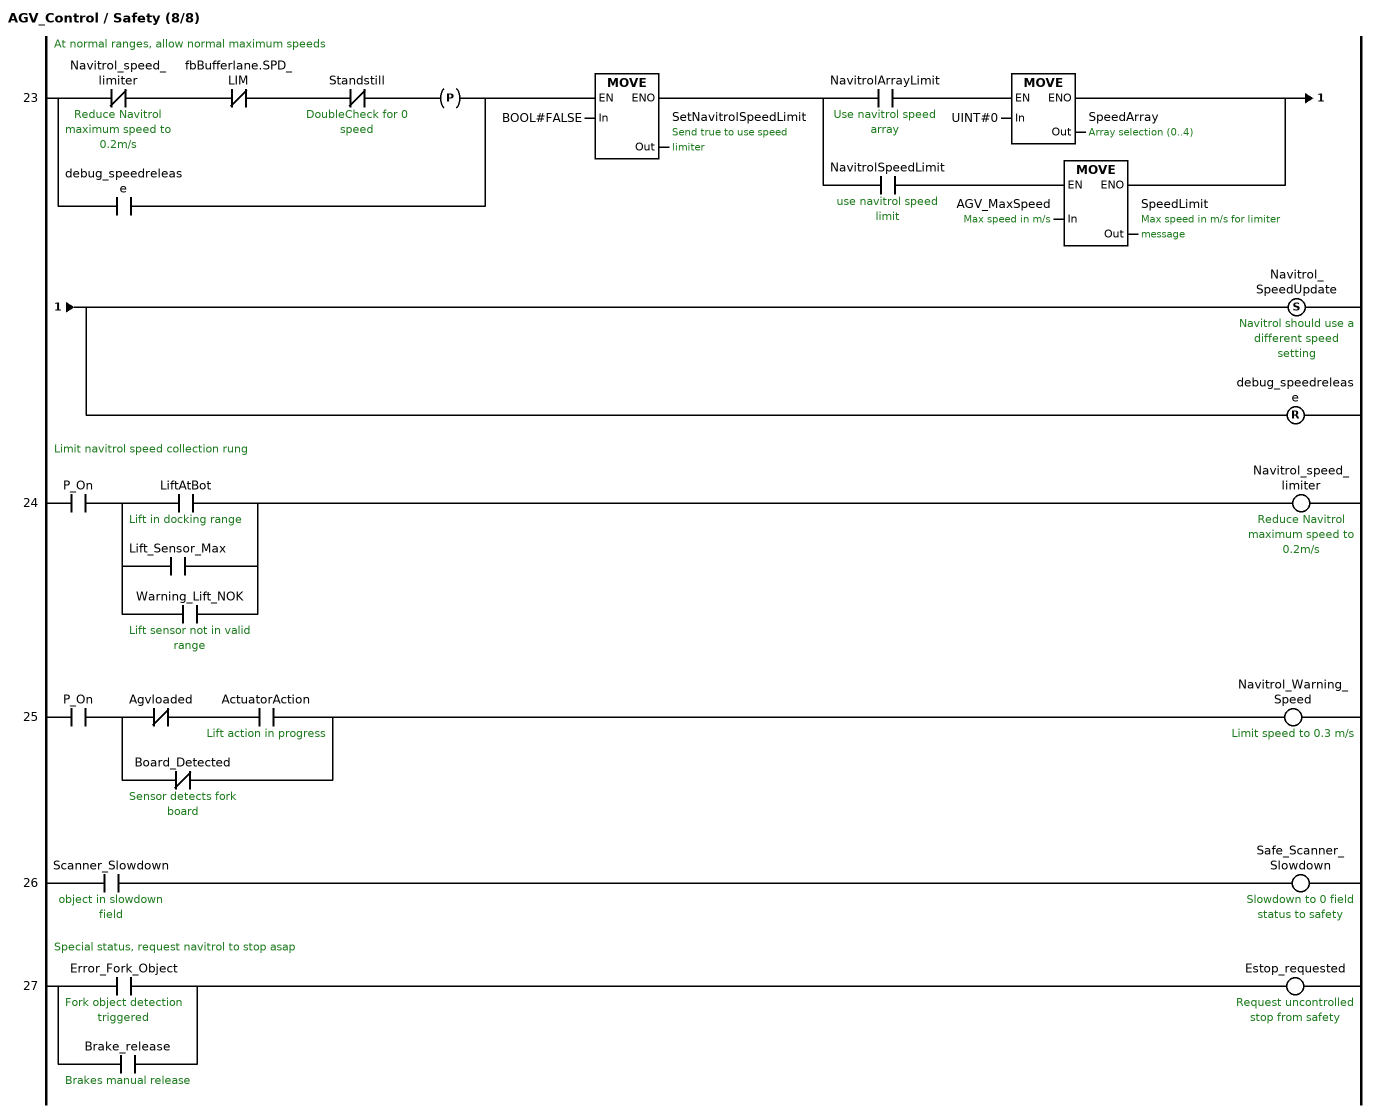
(* Rung 23: At normal ranges, allow normal maximum speeds *)
_e15(CLK := NOT Navitrol_speed_limiter AND NOT fbBufferlane.SPD_LIM AND NOT Standstill);
IF _e15.Q OR debug_speedrelease THEN SetNavitrolSpeedLimit := BOOL#FALSE; END_IF;
IF (_e15.Q OR debug_speedrelease) AND NavitrolArrayLimit THEN SpeedArray := UINT#0; END_IF;
IF (_e15.Q OR debug_speedrelease) AND NavitrolSpeedLimit THEN SpeedLimit := AGV_MaxSpeed; END_IF;
_p16 := (_e15.Q OR debug_speedrelease) AND (NavitrolArrayLimit OR NavitrolSpeedLimit);
IF _p16 THEN
    Navitrol_SpeedUpdate := TRUE;
    debug_speedrelease := FALSE;
END_IF;
(* Rung 24: Limit navitrol speed collection rung *)
Navitrol_speed_limiter := P_On AND (LiftAtBot OR Lift_Sensor_Max OR Warning_Lift_NOK);
(* Rung 25 *)
Navitrol_Warning_Speed := P_On AND ((NOT Agvloaded AND ActuatorAction) OR NOT Board_Detected);
(* Rung 26 *)
Safe_Scanner_Slowdown := Scanner_Slowdown;
(* Rung 27: Special status, request navitrol to stop asap *)
Estop_requested := Error_Fork_Object OR Brake_release;

(* Section Warning: ladder, written here as Structured Text *)

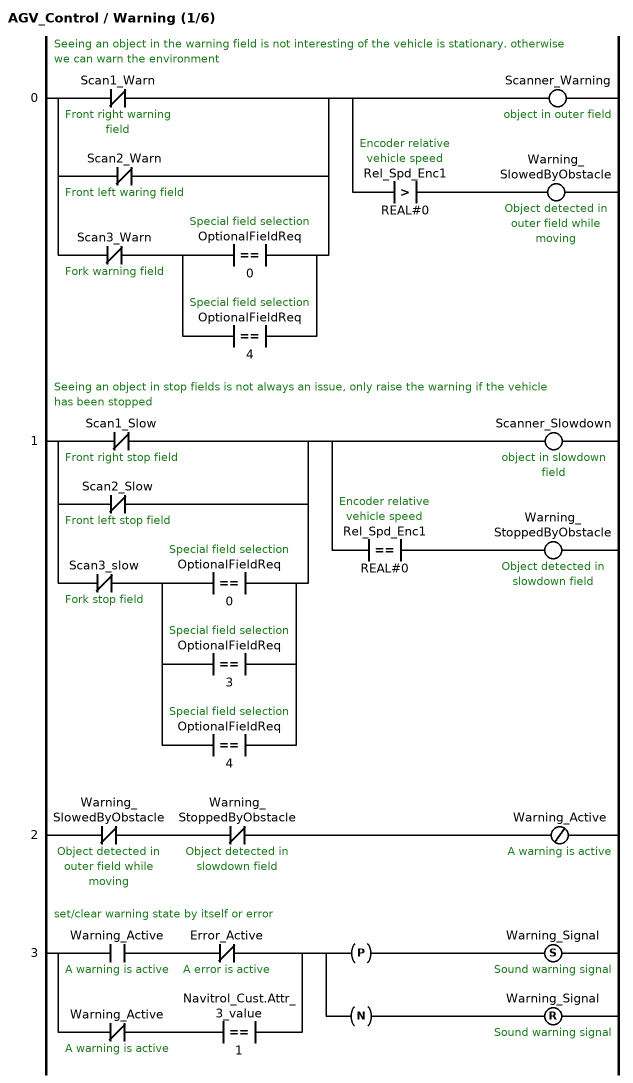
(* Rung 0: Seeing an object in the warning field is not interesting of the vehicle is stationary. otherwise we can warn the environment *)
_p17 := NOT Scan1_Warn OR NOT Scan2_Warn OR (NOT Scan3_Warn AND ((OptionalFieldReq = 0) OR (OptionalFieldReq = 4)));
Scanner_Warning := _p17;
Warning_SlowedByObstacle := _p17 AND (Rel_Spd_Enc1 > REAL#0);
(* Rung 1: Seeing an object in stop fields is not always an issue, only raise the warning if the vehicle has been stopped *)
_p18 := NOT Scan1_Slow OR NOT Scan2_Slow OR (NOT Scan3_slow AND ((OptionalFieldReq = 0) OR (OptionalFieldReq = 3) OR (OptionalFieldReq = 4)));
Scanner_Slowdown := _p18;
Warning_StoppedByObstacle := _p18 AND (Rel_Spd_Enc1 = REAL#0);
(* Rung 2 *)
Warning_Active := NOT (NOT Warning_SlowedByObstacle AND NOT Warning_StoppedByObstacle);
(* Rung 3: set/clear warning state by itself or error *)
_p19 := (Warning_Active AND NOT Error_Active) OR (NOT Warning_Active AND (Navitrol_Cust.Attr_3_value = 1));
_e20(CLK := _p19);
IF _e20.Q THEN Warning_Signal := TRUE; END_IF;
_e21(CLK := _p19);
IF _e21.Q THEN Warning_Signal := FALSE; END_IF;

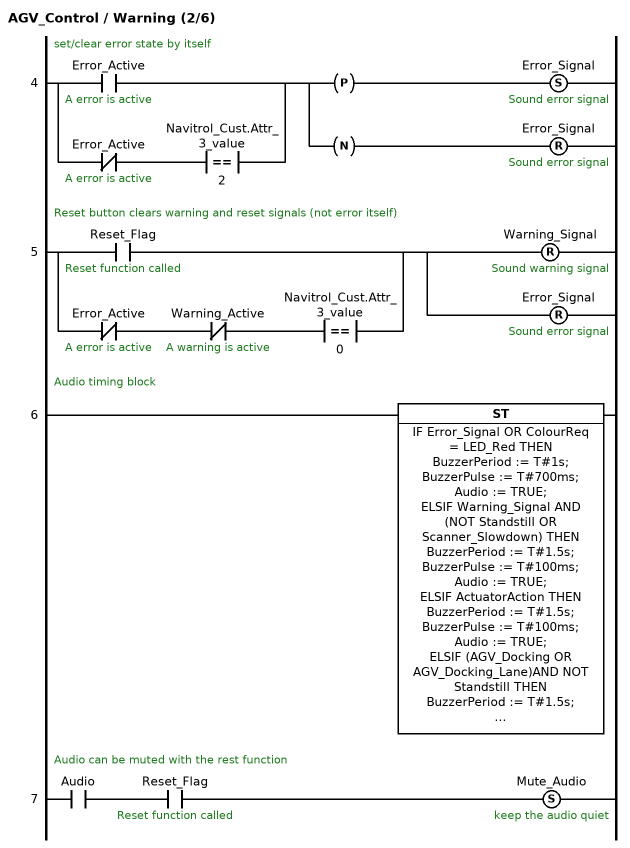
(* Rung 4: set/clear error state by itself *)
_p22 := Error_Active OR (NOT Error_Active AND (Navitrol_Cust.Attr_3_value = 2));
_e23(CLK := _p22);
IF _e23.Q THEN Error_Signal := TRUE; END_IF;
_e24(CLK := _p22);
IF _e24.Q THEN Error_Signal := FALSE; END_IF;
(* Rung 5: Reset button clears warning and reset signals (not error itself) *)
_p25 := Reset_Flag OR (NOT Error_Active AND NOT Warning_Active AND (Navitrol_Cust.Attr_3_value = 0));
IF _p25 THEN
    Warning_Signal := FALSE;
    Error_Signal := FALSE;
END_IF;
(* Rung 6: Audio timing block *)
IF Error_Signal OR ColourReq = LED_Red THEN
	BuzzerPeriod := T#1s;
	BuzzerPulse := T#700ms;
	Audio := TRUE;
ELSIF Warning_Signal AND (NOT Standstill OR Scanner_Slowdown) THEN
	BuzzerPeriod := T#1.5s;
	BuzzerPulse := T#100ms;
	Audio := TRUE;
ELSIF ActuatorAction THEN
	BuzzerPeriod := T#1.5s;
	BuzzerPulse := T#100ms;
	Audio := TRUE;
ELSIF (AGV_Docking OR AGV_Docking_Lane)AND NOT Standstill THEN
	BuzzerPeriod := T#1.5s;
	BuzzerPulse := T#100ms;
	Audio := TRUE;
ELSIF NearTarget_No_Load = TRUE AND MES_Target.Cargo_Required = TRUE then
	BuzzerPeriod := T#1.5s;
	BuzzerPulse := T#100ms;
	Audio := TRUE;
//ELSEIF (fbOverhangDetection)
//
ELSE
	Audio := FALSE;
END_IF;
(* Rung 7: Audio can be muted with the rest function *)
IF Audio AND Reset_Flag THEN Mute_Audio := TRUE; END_IF;

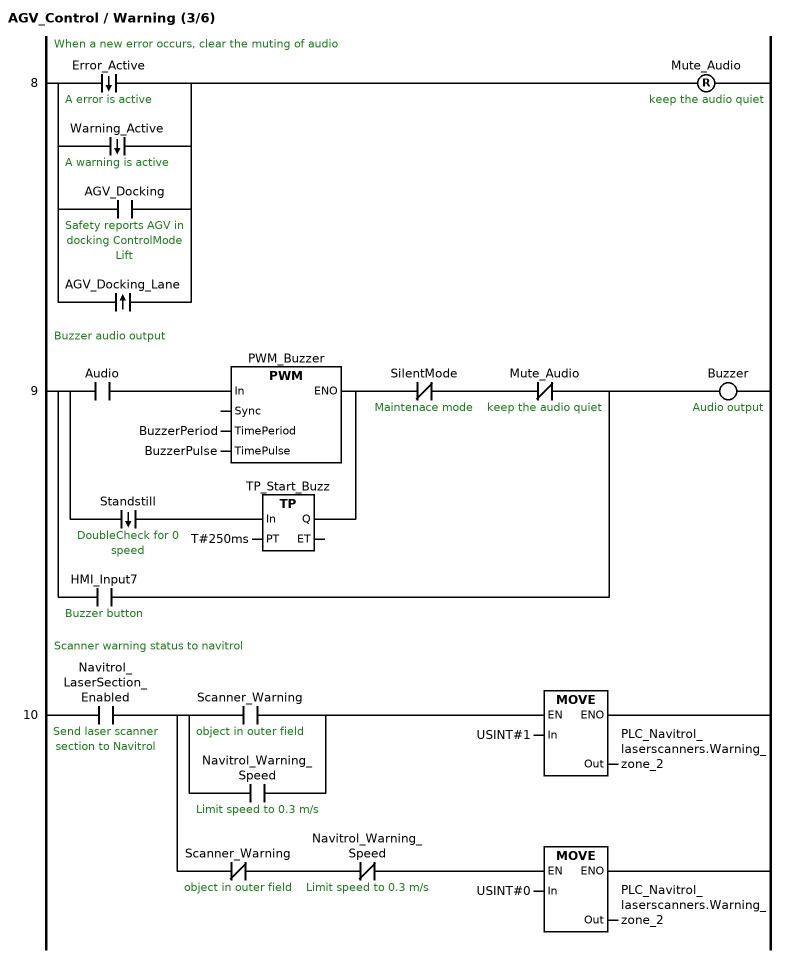
(* Rung 8: When a new error occurs, clear the muting of audio *)
_e26(CLK := Error_Active);
_e27(CLK := Warning_Active);
_e28(CLK := AGV_Docking_Lane);
IF _e26.Q OR _e27.Q OR AGV_Docking OR _e28.Q THEN Mute_Audio := FALSE; END_IF;
(* Rung 9: Buzzer audio output *)
PWM_Buzzer(In := Audio, TimePeriod := BuzzerPeriod, TimePulse := BuzzerPulse);
_e29(CLK := Standstill);
TP_Start_Buzz(In := _e29.Q, PT := T#250ms);
Buzzer := ((PWM_Buzzer.ENO OR TP_Start_Buzz.Q) AND NOT SilentMode AND NOT Mute_Audio) OR HMI_Input7;
(* Rung 10: Scanner warning status to navitrol *)
IF Navitrol_LaserSection_Enabled AND (Scanner_Warning OR Navitrol_Warning_Speed) THEN
    PLC_Navitrol_laserscanners.Warning_zone_2 := USINT#1;
END_IF;
IF Navitrol_LaserSection_Enabled AND NOT Scanner_Warning AND NOT Navitrol_Warning_Speed THEN
    PLC_Navitrol_laserscanners.Warning_zone_2 := USINT#0;
END_IF;

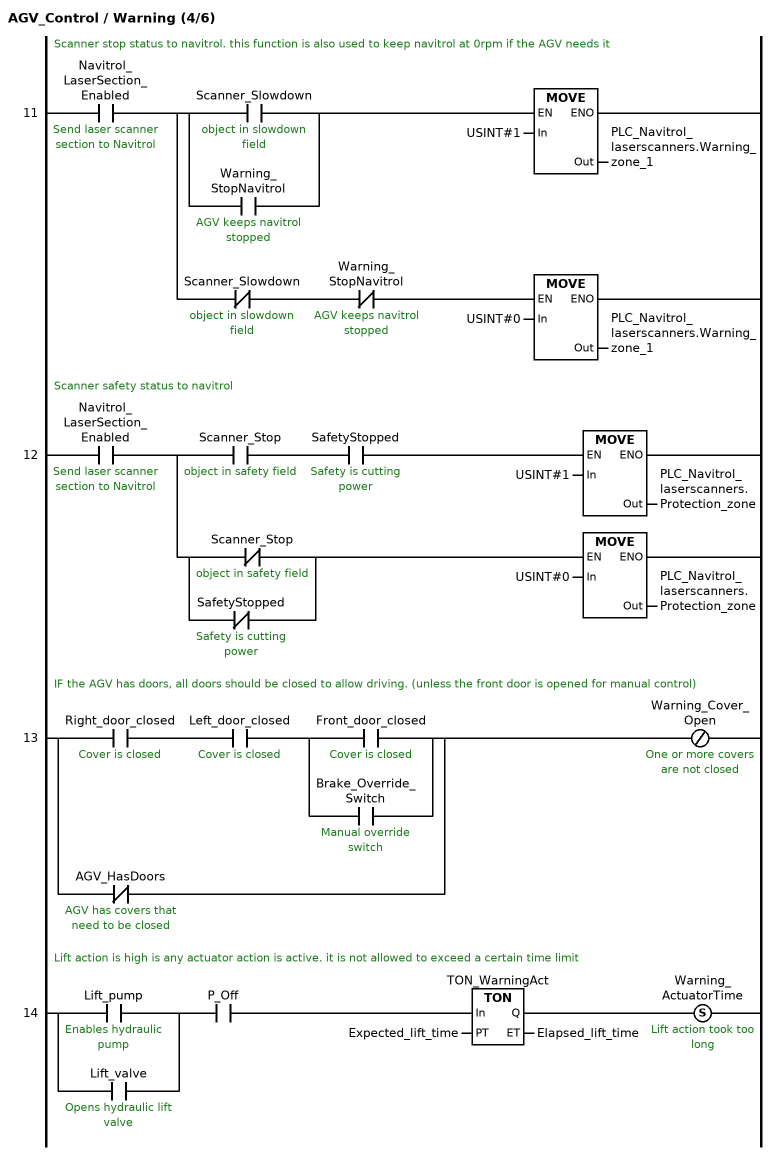
(* Rung 11: Scanner stop status to navitrol. this function is also used to keep navitrol at 0rpm if the AGV needs it *)
IF Navitrol_LaserSection_Enabled AND (Scanner_Slowdown OR Warning_StopNavitrol) THEN
    PLC_Navitrol_laserscanners.Warning_zone_1 := USINT#1;
END_IF;
IF Navitrol_LaserSection_Enabled AND NOT Scanner_Slowdown AND NOT Warning_StopNavitrol THEN
    PLC_Navitrol_laserscanners.Warning_zone_1 := USINT#0;
END_IF;
(* Rung 12: Scanner safety status to navitrol *)
IF Navitrol_LaserSection_Enabled AND Scanner_Stop AND SafetyStopped THEN
    PLC_Navitrol_laserscanners.Protection_zone := USINT#1;
END_IF;
IF Navitrol_LaserSection_Enabled AND (NOT Scanner_Stop OR NOT SafetyStopped) THEN
    PLC_Navitrol_laserscanners.Protection_zone := USINT#0;
END_IF;
(* Rung 13: IF the AGV has doors, all doors should be closed to allow driving. (unless the front door is opened for manual control) *)
Warning_Cover_Open := NOT ((Right_door_closed AND Left_door_closed AND (Front_door_closed OR Brake_Override_Switch)) OR NOT AGV_HasDoors);
(* Rung 14: Lift action is high is any actuator action is active. it is not allowed to exceed a certain time limit *)
TON_WarningAct(In := (Lift_pump OR Lift_valve) AND P_Off, PT := Expected_lift_time, ET => Elapsed_lift_time);
IF TON_WarningAct.Q THEN Warning_ActuatorTime := TRUE; END_IF;

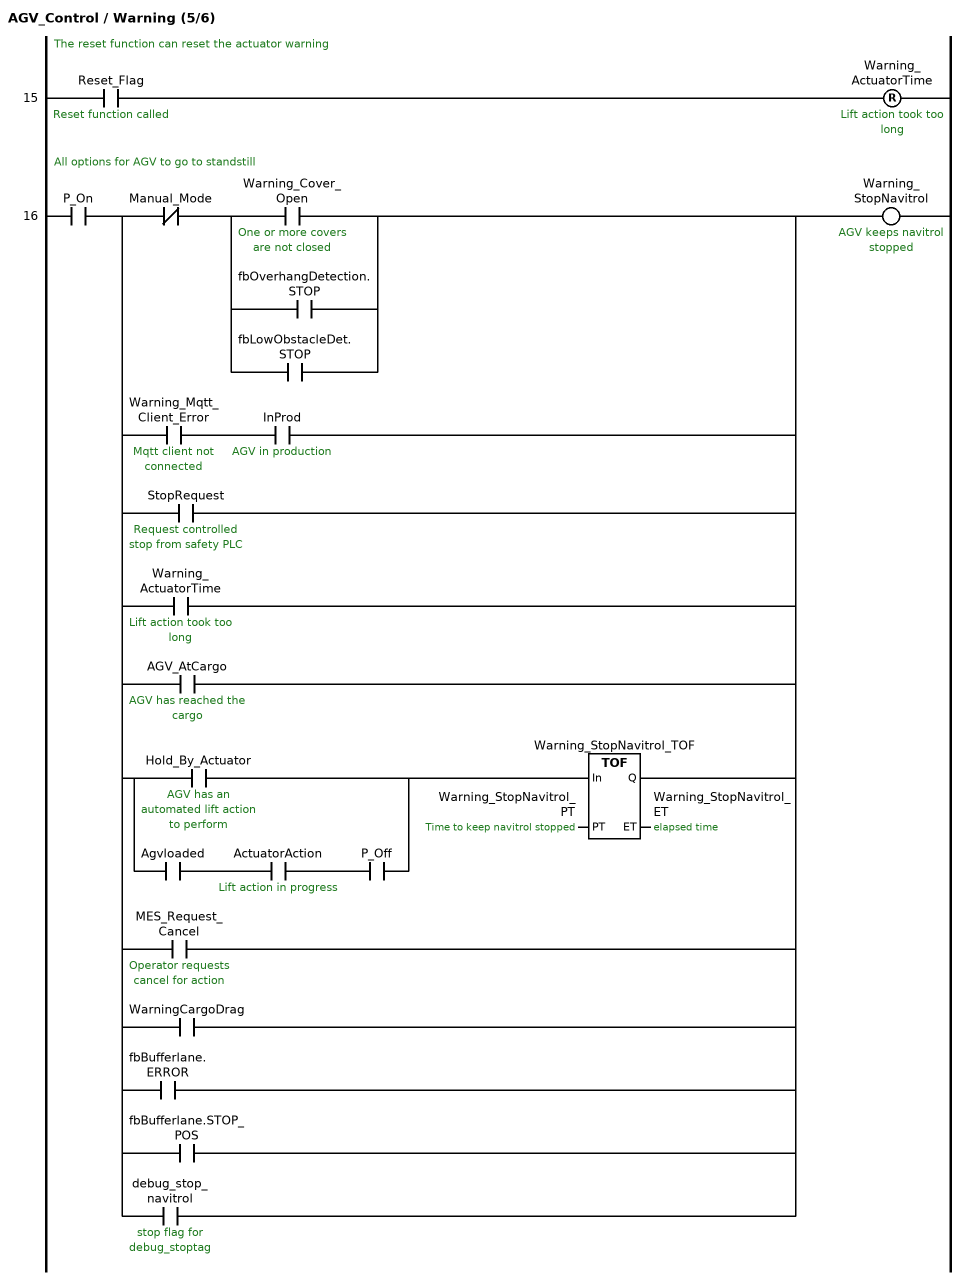
(* Rung 15: The reset function can reset the actuator warning *)
IF Reset_Flag THEN Warning_ActuatorTime := FALSE; END_IF;
(* Rung 16: All options for AGV to go to standstill *)
Warning_StopNavitrol_TOF(In := P_On AND (Hold_By_Actuator OR (Agvloaded AND ActuatorAction AND P_Off)), PT := Warning_StopNavitrol_PT, ET => Warning_StopNavitrol_ET);
Warning_StopNavitrol := (P_On AND ((NOT Manual_Mode AND (Warning_Cover_Open OR fbOverhangDetection.STOP OR fbLowObstacleDet.STOP)) OR (Warning_Mqtt_Client_Error AND InProd) OR StopRequest OR Warning_ActuatorTime OR AGV_AtCargo)) OR Warning_StopNavitrol_TOF.Q OR (P_On AND (MES_Request_Cancel OR WarningCargoDrag OR fbBufferlane.ERROR OR fbBufferlane.STOP_POS OR debug_stop_navitrol));

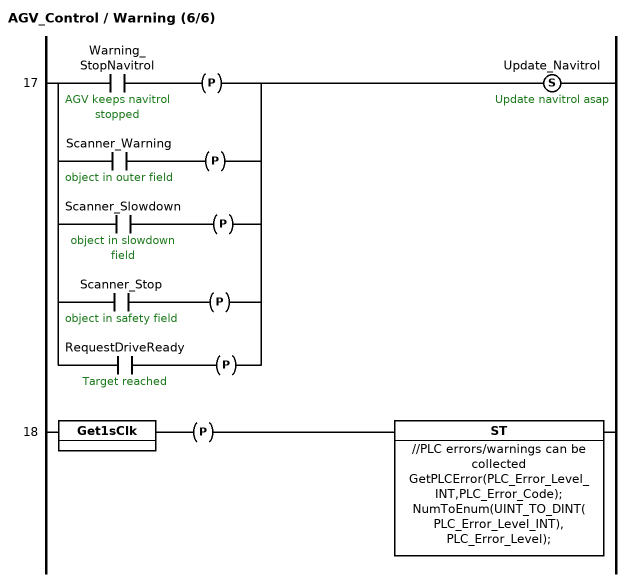
(* Rung 17 *)
_e30(CLK := Warning_StopNavitrol);
_e31(CLK := Scanner_Warning);
_e32(CLK := Scanner_Slowdown);
_e33(CLK := Scanner_Stop);
_e34(CLK := RequestDriveReady);
IF _e30.Q OR _e31.Q OR _e32.Q OR _e33.Q OR _e34.Q THEN Update_Navitrol := TRUE; END_IF;
(* Rung 18 *)
_e35(CLK := Get1sClk());
IF _e35.Q THEN
    //PLC errors/warnings can be collected
    GetPLCError(PLC_Error_Level_INT,PLC_Error_Code);
    NumToEnum(UINT_TO_DINT(PLC_Error_Level_INT), PLC_Error_Level);
END_IF;

(* Section LEDs: ladder, written here as Structured Text *)

